//*************************************************************************************FORCE COLOR & BRIGHTNESS - LEVEL
IF sDeviceType = Domoticz_Constants.sType_LightSwitch
AND xForceSetValues
AND NOT xFading_int
	//Brightness	
AND ((NOT _Domoticz_EqualWithWindow(byBrightness_int, scColorData_Act.byBrightness, 5) AND xEnable_int)
	OR (NOT _Domoticz_EqualWithWindow(byBrightness_int, scColorData_Act.byBrightness, 1) AND (byBrightness_int = 0 OR NOT xEnable_int))) 
THEN
	
	//Set mode
	afb_ObjectArrayReal_InOut[1].eCommandType := _Domoticz_eCommandType.SetBrightness;	//Don't use default uDevice
	
	//Transfer outgoing data
	afb_ObjectArrayReal_InOut[1].arValueSet[Domoticz_eSValues_Colors.Brightness]:= _Domoticz_RoundDecimals(((TO_REAL(byBrightness_int)/255)*100),0);

	//Force
	afb_ObjectArrayReal_InOut[1].ForceSet(tForceSetValues_int);

//*************************************************************************************FORCE COLOR & BRIGHTNESS - COLOR SWITCH
ELSIF sDeviceType = Domoticz_Constants.sType_ColorSwitch
AND xForceSetValues
AND NOT xFading_int
AND (NOT xColorActValid OR NOT xEnable_int OR (xEnable_int AND NOT xEnabled))
	//Brightness	
AND ((NOT _Domoticz_EqualWithWindow(byBrightness_int, scColorData_Act.byBrightness, 5) AND xEnable_int)
	OR (NOT _Domoticz_EqualWithWindow(byBrightness_int, scColorData_Act.byBrightness, 1) AND (byBrightness_int = 0 OR NOT xEnable_int))
	//Colors
	OR (NOT _Domoticz_EqualWithWindow(scColorData_Set.byRed, scColorData_Act.byRed, 1) AND xEnable_int)
	OR (NOT _Domoticz_EqualWithWindow(scColorData_Set.byGreen, scColorData_Act.byGreen, 1) AND xEnable_int)
	OR (NOT _Domoticz_EqualWithWindow(scColorData_Set.byBlue, scColorData_Act.byBlue, 1) AND xEnable_int)
	//Temperature
	OR (NOT _Domoticz_EqualWithWindow(scColorData_Set.byColdWhite, scColorData_Act.byColdWhite, 1) AND xEnable_int)
	OR (NOT _Domoticz_EqualWithWindow(scColorData_Set.byWarmWhite, scColorData_Act.byWarmWhite, 1) AND xEnable_int)) 
THEN
	
	//Set mode
	afb_ObjectArrayReal_InOut[1].eCommandType := _Domoticz_eCommandType.SetColor;	//Don't use default uDevice
	
	//Transfer outgoing data
	afb_ObjectArrayReal_InOut[1].arValueSet[Domoticz_eSValues_Colors.Brightness]:= _Domoticz_RoundDecimals(((TO_REAL(byBrightness_int)/255)*100),0);
	afb_ObjectArrayReal_InOut[1].arValueSet[Domoticz_eSValues_Colors.Red]		:= TO_REAL(scColorData_Set.byRed);
	afb_ObjectArrayReal_InOut[1].arValueSet[Domoticz_eSValues_Colors.Green]	:= TO_REAL(scColorData_Set.byGreen);
	afb_ObjectArrayReal_InOut[1].arValueSet[Domoticz_eSValues_Colors.Blue]		:= TO_REAL(scColorData_Set.byBlue);
	afb_ObjectArrayReal_InOut[1].arValueSet[Domoticz_eSValues_Colors.ColdWhite] := TO_REAL(scColorData_Set.byColdWhite);
	afb_ObjectArrayReal_InOut[1].arValueSet[Domoticz_eSValues_Colors.WarmWhite] := TO_REAL(scColorData_Set.byWarmWhite);

	//Force
	afb_ObjectArrayReal_InOut[1].ForceSet(tForceSetValues_int);
END_IF

//*************************************************************************************ERRORS
fbEI_DataTimeOut.sInstanceName := sInstanceName;
fbEI_DataTimeOut.tErrorDelay := T#500MS;	//Give objects TIME TO be overruled BY other updates
fbEI_DataTimeOut(
	scConnector:= scConnector,
	xError:= xDataTimeOut_int
			AND (afb_ObjectArrayReal_InOut[1].xDataTimedOut),
	eErrorID:= Domoticz_eErrors.ObjectDataTimeOut
);
END_ACTION

{attribute 'monitoring' := 'call'} PROPERTY tFadeTime :TIME
GET
tFadeTime := tFadeTime_int;
END_GET
SET
tFadeTime_int := tFadeTime;
END_SET
END_PROPERTY

{attribute 'monitoring' := 'call'} PROPERTY tFadeUpdateTime :TIME
SET
tFadeUpdateTime_int := tFadeUpdateTime;
END_SET
GET
tFadeUpdateTime := tFadeUpdateTime_int;
END_GET
END_PROPERTY

{attribute 'monitoring' := 'call'} PROPERTY xFading :BOOL
GET
xFading := xFading_int;
END_GET
END_PROPERTY

END_FUNCTION_BLOCK

// Functions/_Domoticz_EqualWithWindow
{attribute 'conditionalshow_all_locals'}
{attribute 'conditionalshow'}
FUNCTION _Domoticz_EqualWithWindow :BOOL
VAR_INPUT
	rInput1, rInput2, rWindow :REAL;
END_VAR
VAR
END_VAR

_Domoticz_EqualWithWindow := (rInput1 >= (rInput2 - rWindow) AND rInput1 <= (rInput2 + rWindow));

END_FUNCTION

// Functions/_Domoticz_ColorFactor
{attribute 'conditionalshow_all_locals'}
{attribute 'conditionalshow'}
FUNCTION _Domoticz_ColorFactor :REAL
VAR_INPUT
	byColorSet	:BYTE;
	byColorAct	:BYTE;
END_VAR
VAR
END_VAR

IF byColorAct <> 0 AND byColorSet <> 0 THEN
	_Domoticz_ColorFactor := TO_REAL(byColorAct)/TO_REAL(byColorSet);
ELSIF byColorAct <> 0 AND byColorSet = 0 THEN
	_Domoticz_ColorFactor := -255;
ELSIF byColorAct = 0 AND byColorSet <> 0 THEN
	_Domoticz_ColorFactor := 255;
ELSE
	_Domoticz_ColorFactor := 0;
END_IF

END_FUNCTION

// Function Blocks/Hardware/Weather/Domoticz_AccuWeather
{attribute 'conditionalshow_all_locals'}
FUNCTION_BLOCK Domoticz_AccuWeather EXTENDS _Domoticz_Connector_Out
VAR_INPUT
	uiIdentifier_TempHumBaro	:UINT;	//Temperature/humidity/barometer
	uiIdentifier_Rain			:UINT;	//Rain rate and actual
	uiIdentifier_Wind			:UINT;	//Wind (direction,strenght)
	uiIdentifier_Visibility		:UINT;	//Visibility outside
	uiIdentifier_UV				:UINT;	//UV power
END_VAR
VAR_OUTPUT
	rTemperature				:REAL;
	rDewPoint					:REAL;
	rChill						:REAL;
	rHumidity					:REAL;
	rBaroMeter					:REAL;
	rRain						:REAL;
	rRainRate					:REAL;
	rWindSpeed					:REAL;
	rWindGust					:REAL;
	rWindDirection				:REAL;
	rVisibility					:REAL;
	rUV							:REAL;
END_VAR
VAR
	afb_ObjectArrayReal_Out		:ARRAY[1..3] OF _Domoticz_ObjectArrayReal_Out;
	afb_ObjectReal_Out			:ARRAY[1..2] OF _Domoticz_ObjectReal_Out;
END_VAR

IF __ISVALIDREF(scConnector) THEN
	Main();
END_IF

ACTION Main:
{attribute 'conditionalshow'}
//Call parent function
SUPER^.Main();

//Call all functions
//Extended data timeout (Weather not updated frequently)
afb_ObjectArrayReal_Out[1].tDataTimeOut := T#24H;
afb_ObjectArrayReal_Out[1](	scConnector := scConnector, 	uiIdentifier := uiIdentifier_TempHumBaro,	rxUpdateInterlock := rxUpdateInterlock_int);
                                                            
afb_ObjectArrayReal_Out[2].tDataTimeOut := T#24H;           
afb_ObjectArrayReal_Out[2](	scConnector := scConnector, 	uiIdentifier := uiIdentifier_Wind,			rxUpdateInterlock := rxUpdateInterlock_int);
                                                            
afb_ObjectArrayReal_Out[3].tDataTimeOut := T#24H;           
afb_ObjectArrayReal_Out[3](	scConnector := scConnector,		uiIdentifier := uiIdentifier_Rain,			rxUpdateInterlock := rxUpdateInterlock_int);
                                                            
afb_ObjectReal_Out[1].tDataTimeOut := T#24H;                
afb_ObjectReal_Out[1](		scConnector := scConnector, 	uiIdentifier := uiIdentifier_Visibility,	rxUpdateInterlock := rxUpdateInterlock_int,		rValueAct => rVisibility);
                                                            
afb_ObjectReal_Out[2].tDataTimeOut := T#24H;                
afb_ObjectReal_Out[2](		scConnector := scConnector, 	uiIdentifier := uiIdentifier_UV,			rxUpdateInterlock := rxUpdateInterlock_int,		rValueAct => rUV);

//Output arrays
rTemperature 	:= afb_ObjectArrayReal_Out[1].arValueAct[Domoticz_eSValues_TempHumBaro.Temperature];
rDewPoint		:= afb_ObjectArrayReal_Out[1].arValueAct[Domoticz_eSValues_TempHumBaro.DewPoint];
rHumidity		:= afb_ObjectArrayReal_Out[1].arValueAct[Domoticz_eSValues_TempHumBaro.Humidity];
rBaroMeter		:= afb_ObjectArrayReal_Out[1].arValueAct[Domoticz_eSValues_TempHumBaro.Barometer];

rWindSpeed	 	:= afb_ObjectArrayReal_Out[2].arValueAct[Domoticz_eSValues_Wind.Speed];
rChill			:= afb_ObjectArrayReal_Out[2].arValueAct[Domoticz_eSValues_Wind.Chill];
rWindGust		:= afb_ObjectArrayReal_Out[2].arValueAct[Domoticz_eSValues_Wind.Gust];
rWindDirection	:= afb_ObjectArrayReal_Out[2].arValueAct[Domoticz_eSValues_Wind.Bearing];

rRain		 	:= afb_ObjectArrayReal_Out[3].arValueAct[Domoticz_eSValues_Rain.Rain];
rRainRate		:= afb_ObjectArrayReal_Out[3].arValueAct[Domoticz_eSValues_Rain.RainRate];

//Errors
fbEI_DataTimeOut.sInstanceName := sInstanceName;
fbEI_DataTimeOut.tErrorDelay := T#500MS;	//Give objects TIME TO be overruled BY other updates
fbEI_DataTimeOut(
	scConnector:= scConnector,
	xError:= xDataTimeOut_int
			AND (afb_ObjectArrayReal_Out[1].xDataTimedOut
			OR afb_ObjectArrayReal_Out[2].xDataTimedOut
			OR afb_ObjectArrayReal_Out[3].xDataTimedOut
			OR afb_ObjectReal_Out[1].xDataTimedOut
			OR afb_ObjectReal_Out[2].xDataTimedOut),
	eErrorID:= Domoticz_eErrors.ObjectDataTimeOut
);
END_ACTION

END_FUNCTION_BLOCK

// Function Blocks/Hardware/Weather/Domoticz_BuienAlarm
{attribute 'conditionalshow_all_locals'}
FUNCTION_BLOCK Domoticz_BuienAlarm EXTENDS _Domoticz_Connector_Out
VAR_INPUT
	uiIdentifier_Rain			:UINT;	//Rain rate and actual
	uiIdentifier_RainAlert		:UINT;	//Rain alert
	uiIdentifier_RainForecast	:UINT;	//Rain forecast
END_VAR
VAR_OUTPUT
	rRain						:REAL;
	rRainRate					:REAL;
	rRainForecast				:REAL;
	sRainAlert					:STRING(Domoticz_Constants.uiMaxSValuesize);
	sRainForecast				:STRING(Domoticz_Constants.uiMaxSValuesize);
END_VAR
VAR
	afb_ObjectArrayReal_Out		:ARRAY[1..1] OF _Domoticz_ObjectArrayReal_Out;
	afb_ObjectString_Out		:ARRAY[1..2] OF _Domoticz_ObjectString_Out;
END_VAR

IF __ISVALIDREF(scConnector) THEN
	Main();
END_IF

ACTION Main:
{attribute 'conditionalshow'}
//Call parent function
SUPER^.Main();

//Call all functions
//Extended data timeout, expect a litle rain at least once every two weeks.
afb_ObjectArrayReal_Out[1].tDataTimeOut := T#14D;
afb_ObjectArrayReal_Out[1].eDataSource := _Domoticz_eDataSource.HTTP;  
afb_ObjectArrayReal_Out[1](	scConnector := scConnector, 	uiIdentifier := uiIdentifier_Rain,			rxUpdateInterlock := rxUpdateInterlock_int);
                                                                                                                                                                                  
afb_ObjectString_Out[1].tDataTimeOut := T#14D;      
afb_ObjectString_Out[1].eDataSource := _Domoticz_eDataSource.HTTP;                                                                              
afb_ObjectString_Out[1](	scConnector := scConnector, 	uiIdentifier := uiIdentifier_RainAlert, 	rxUpdateInterlock := rxUpdateInterlock_int,			sValueAct => sRainAlert);
                                                                                                                                                                                
afb_ObjectString_Out[2].tDataTimeOut := T#14D; 
afb_ObjectString_Out[2].eDataSource := _Domoticz_eDataSource.HTTP;                                                                                                              
afb_ObjectString_Out[2](	scConnector := scConnector, 	uiIdentifier := uiIdentifier_RainForecast, 	rxUpdateInterlock := rxUpdateInterlock_int,			sValueAct => sRainForecast);

//Output arrays
rRain		 	:= afb_ObjectArrayReal_Out[1].arValueAct[Domoticz_eSValues_Rain.Rain];
rRainRate		:= afb_ObjectArrayReal_Out[1].arValueAct[Domoticz_eSValues_Rain.RainRate];
rRainForecast	:= _Domoticz_StringToReal(sRainAlert);

//Errors
fbEI_DataTimeOut.sInstanceName := sInstanceName;
fbEI_DataTimeOut.tErrorDelay := T#500MS;	//Give objects TIME TO be overruled BY other updates
fbEI_DataTimeOut(
	scConnector:= scConnector,
	xError:= xDataTimeOut_int
			AND (afb_ObjectArrayReal_Out[1].xDataTimedOut
			OR afb_ObjectString_Out[1].xDataTimedOut
			OR afb_ObjectString_Out[2].xDataTimedOut),
	eErrorID:= Domoticz_eErrors.ObjectDataTimeOut
);
END_ACTION

END_FUNCTION_BLOCK

// Function Blocks/Hardware/Weather/Domoticz_BuienRadar
{attribute 'conditionalshow_all_locals'}
FUNCTION_BLOCK Domoticz_BuienRadar EXTENDS _Domoticz_Connector_Out
VAR_INPUT
	uiIdentifier_TempHumBaro		:UINT;	//Temperature/humidity/barometer
	uiIdentifier_TempGround			:UINT;	//Ground temperature
	uiIdentifier_TempFeel			:UINT;	//Feel temperature
	uiIdentifier_Wind				:UINT;	//Wind (direction,strenght)	
	uiIdentifier_Visibility			:UINT;	//Visibility outside
	uiIdentifier_Solar				:UINT;	//Solar power
	uiIdentifier_Rain				:UINT;	//Rain
	uiIdentifier_RainNextHour		:UINT;	//Rain forecast next hour
	uiIdentifier_RainIntensity		:UINT;	//Rain intensity
	uiIdentifier_RainingMeasured	:UINT;	//Raining - measured at weather station
	uiIdentifier_RainingForecast	:UINT;	//Raining - forecasted at current location
	uiIdentifier_NextRainTime		:UINT;	//Next rainshower time
	uiIdentifier_NextRainDuration	:UINT;	//Next rainshower duration
	uiIdentifier_NextRainAvgRate	:UINT;	//Next rainshower avg rate
	uiIdentifier_NextRainMaxRate	:UINT;	//Next rainshower max rate
END_VAR
VAR_OUTPUT
	rTemperature					:REAL;
	rTemperatureGround				:REAL;
	rTemperatureFeel				:REAL;
	rHumidity						:REAL;
	rBaroMeter						:REAL;
	rWindSpeed						:REAL;
	rWindGust						:REAL;
	rWindDirection					:REAL;
	rVisibility						:REAL;
	rSolar							:REAL;
	rRain							:REAL;
	rRainRate						:REAL;
	rRainNextHour					:REAL;
	rRainIntensity					:REAL;
	xRainingMeasured				:BOOL;
	xRainingForecast				:BOOL;
	tNextRainTime					:TIME;
	tNextRainDuration				:TIME;
	rNextRainAvgRate				:REAL;
	rNextRainMaxRate				:REAL;
END_VAR                         	
VAR                             	
	afb_ObjectArrayReal_Out			:ARRAY[1..3] OF _Domoticz_ObjectArrayReal_Out;
	afb_ObjectReal_Out				:ARRAY[1..10] OF _Domoticz_ObjectReal_Out;
	afb_ObjectBool_Out				:ARRAY[1..2] OF _Domoticz_ObjectBool_Out;
END_VAR

IF __ISVALIDREF(scConnector) THEN
	Main();
END_IF

ACTION Main:
{attribute 'conditionalshow'}
//Call parent function
SUPER^.Main();

//Call all functions
//Extended data timeout (Weather not updated frequently)
afb_ObjectArrayReal_Out[1].tDataTimeOut := T#24H;
afb_ObjectArrayReal_Out[1].eDataSource := _Domoticz_eDataSource.HTTP;
afb_ObjectArrayReal_Out[1](	scConnector := scConnector, 	uiIdentifier := uiIdentifier_TempHumBaro,		rxUpdateInterlock := rxUpdateInterlock_int);
                                                                                                                                                
afb_ObjectArrayReal_Out[2].tDataTimeOut := T#24H;    
afb_ObjectArrayReal_Out[2].eDataSource := _Domoticz_eDataSource.HTTP;                                                                                           
afb_ObjectArrayReal_Out[2](	scConnector := scConnector, 	uiIdentifier := uiIdentifier_Rain,				rxUpdateInterlock := rxUpdateInterlock_int);
                                                                                             
afb_ObjectArrayReal_Out[3].tDataTimeOut := T#24H;                                            
afb_ObjectArrayReal_Out[3].eDataSource := _Domoticz_eDataSource.HTTP;                                 
afb_ObjectArrayReal_Out[3](	scConnector := scConnector, 	uiIdentifier := uiIdentifier_Wind,				rxUpdateInterlock := rxUpdateInterlock_int);
                                                                                                                                                
afb_ObjectReal_Out[1].tDataTimeOut := T#24H;  
afb_ObjectReal_Out[1].eDataSource := _Domoticz_eDataSource.HTTP;                                                                                                  
afb_ObjectReal_Out[1](		scConnector := scConnector, 	uiIdentifier := uiIdentifier_TempGround,		rxUpdateInterlock := rxUpdateInterlock_int,			rValueAct => rTemperatureGround);
                                                                                                                                            
afb_ObjectReal_Out[2].tDataTimeOut := T#24H;                                                                                                
afb_ObjectReal_Out[2].eDataSource := _Domoticz_eDataSource.HTTP;                                                                                           
afb_ObjectReal_Out[2](		scConnector := scConnector, 	uiIdentifier := uiIdentifier_TempFeel,			rxUpdateInterlock := rxUpdateInterlock_int,			rValueAct => rTemperatureFeel);
                                                                                                                                            
afb_ObjectReal_Out[3].tDataTimeOut := T#24H;                                                                                                
afb_ObjectReal_Out[3].eDataSource := _Domoticz_eDataSource.HTTP;                                                                                           
afb_ObjectReal_Out[3](		scConnector := scConnector, 	uiIdentifier := uiIdentifier_Visibility,		rxUpdateInterlock := rxUpdateInterlock_int,			rValueAct => rVisibility);
                                                                                                                                            
afb_ObjectReal_Out[4].tDataTimeOut := T#24H;                                                                                                
afb_ObjectReal_Out[4].eDataSource := _Domoticz_eDataSource.HTTP;                                                                                               
afb_ObjectReal_Out[4](		scConnector := scConnector, 	uiIdentifier := uiIdentifier_Solar,				rxUpdateInterlock := rxUpdateInterlock_int,			rValueAct => rSolar);
                                                                                                                                            
afb_ObjectReal_Out[5].tDataTimeOut := T#24H;                                                                                                
afb_ObjectReal_Out[5].eDataSource := _Domoticz_eDataSource.HTTP;                                                                                              
afb_ObjectReal_Out[5](		scConnector := scConnector, 	uiIdentifier := uiIdentifier_RainNextHour,		rxUpdateInterlock := rxUpdateInterlock_int,			rValueAct => rRainNextHour);
                                                                                                                                            
afb_ObjectReal_Out[6].tDataTimeOut := T#24H;                                                                                                
afb_ObjectReal_Out[6].eDataSource := _Domoticz_eDataSource.HTTP;                                                                                              
afb_ObjectReal_Out[6](		scConnector := scConnector, 	uiIdentifier := uiIdentifier_RainIntensity,		rxUpdateInterlock := rxUpdateInterlock_int,			rValueAct => rRainIntensity);
                                                                                                                                                                                           
afb_ObjectReal_Out[7].tDataTimeOut := T#24H;      
afb_ObjectReal_Out[7].eDataSource := _Domoticz_eDataSource.HTTP;                                                                                                                                         
afb_ObjectReal_Out[7](		scConnector := scConnector, 	uiIdentifier := uiIdentifier_NextRainTime,		rxUpdateInterlock := rxUpdateInterlock_int);                             
                                                                                                                                           
afb_ObjectReal_Out[8].tDataTimeOut := T#24H;                                                                
afb_ObjectReal_Out[8].eDataSource := _Domoticz_eDataSource.HTTP;                                                                                          
afb_ObjectReal_Out[8](		scConnector := scConnector, 	uiIdentifier := uiIdentifier_NextRainDuration,	rxUpdateInterlock := rxUpdateInterlock_int);                             
                                                                                                                                                                                           
afb_ObjectReal_Out[9].tDataTimeOut := T#24H;                                                                                                                                               
afb_ObjectReal_Out[9].eDataSource := _Domoticz_eDataSource.HTTP;
afb_ObjectReal_Out[9](		scConnector := scConnector, 	uiIdentifier := uiIdentifier_NextRainAvgRate,	rxUpdateInterlock := rxUpdateInterlock_int,			rValueAct => rNextRainAvgRate);
                                                                                                                                         
afb_ObjectReal_Out[10].tDataTimeOut := T#24H;                                                                                            
afb_ObjectReal_Out[10].eDataSource := _Domoticz_eDataSource.HTTP;                                                                                        
afb_ObjectReal_Out[10](		scConnector := scConnector, 	uiIdentifier := uiIdentifier_NextRainMaxRate,	rxUpdateInterlock := rxUpdateInterlock_int,			rValueAct => rNextRainMaxRate);
                                                                                                                                         
afb_ObjectBool_Out[1].tDataTimeOut := T#24H;                                                                                             
afb_ObjectBool_Out[1].eDataSource := _Domoticz_eDataSource.HTTP;                                                                          
afb_ObjectBool_Out[1](		scConnector := scConnector, 	uiIdentifier := uiIdentifier_RainingMeasured,	rxUpdateInterlock := rxUpdateInterlock_int,			xValueAct => xRainingMeasured);
                                                                                                                                         
afb_ObjectBool_Out[2].tDataTimeOut := T#14D;                                                                                             
afb_ObjectBool_Out[2].eDataSource := _Domoticz_eDataSource.HTTP;                                                                                
afb_ObjectBool_Out[2](		scConnector := scConnector, 	uiIdentifier := uiIdentifier_RainingForecast,	rxUpdateInterlock := rxUpdateInterlock_int,			xValueAct => xRainingForecast);


//Output arrays
rTemperature 		:= afb_ObjectArrayReal_Out[1].arValueAct[Domoticz_eSValues_TempHumBaro.Temperature];
rHumidity			:= afb_ObjectArrayReal_Out[1].arValueAct[Domoticz_eSValues_TempHumBaro.Humidity];
rBaroMeter			:= afb_ObjectArrayReal_Out[1].arValueAct[Domoticz_eSValues_TempHumBaro.Barometer];
                		                	
rRain		 		:= afb_ObjectArrayReal_Out[2].arValueAct[Domoticz_eSValues_Rain.Rain];
rRainRate			:= afb_ObjectArrayReal_Out[2].arValueAct[Domoticz_eSValues_Rain.RainRate];

rWindSpeed	 		:= afb_ObjectArrayReal_Out[3].arValueAct[Domoticz_eSValues_Wind.Speed];
rWindGust			:= afb_ObjectArrayReal_Out[3].arValueAct[Domoticz_eSValues_Wind.Gust];
rWindDirection		:= afb_ObjectArrayReal_Out[3].arValueAct[Domoticz_eSValues_Wind.Bearing];
                	
tNextRainTime		:= TO_TIME(afb_ObjectReal_Out[7].rValueAct * 60 * 1000);
tNextRainDuration 	:= TO_TIME(afb_ObjectReal_Out[8].rValueAct * 60 * 1000); 
										   
//Errors
fbEI_DataTimeOut.sInstanceName := sInstanceName;
fbEI_DataTimeOut.tErrorDelay := T#500MS;	//Give objects TIME TO be overruled BY other updates
fbEI_DataTimeOut(
	scConnector:= scConnector,
	xError:= xDataTimeOut_int
			AND (afb_ObjectArrayReal_Out[1].xDataTimedOut
			OR afb_ObjectArrayReal_Out[2].xDataTimedOut
			OR afb_ObjectArrayReal_Out[3].xDataTimedOut
			OR afb_ObjectReal_Out[1].xDataTimedOut
			OR afb_ObjectReal_Out[2].xDataTimedOut
			OR afb_ObjectReal_Out[3].xDataTimedOut
			OR afb_ObjectReal_Out[4].xDataTimedOut
			OR afb_ObjectReal_Out[5].xDataTimedOut
			OR afb_ObjectReal_Out[6].xDataTimedOut
			OR afb_ObjectReal_Out[7].xDataTimedOut
			OR afb_ObjectReal_Out[8].xDataTimedOut
			OR afb_ObjectReal_Out[9].xDataTimedOut
			OR afb_ObjectReal_Out[10].xDataTimedOut
			OR afb_ObjectBool_Out[1].xDataTimedOut
			OR afb_ObjectBool_Out[2].xDataTimedOut),
	eErrorID:= Domoticz_eErrors.ObjectDataTimeOut
);
END_ACTION

END_FUNCTION_BLOCK

// Function Blocks/Hardware/Weather/Domoticz_BuienRadar_Forecast
{attribute 'conditionalshow_all_locals'}
FUNCTION_BLOCK Domoticz_BuienRadar_Forecast EXTENDS _Domoticz_Connector_Out
VAR_INPUT
	uiIdentifier_TempMin		:UINT;	//Minimal temperature
	uiIdentifier_TempMax		:UINT;	//Maixmal temperature
	uiIdentifier_SunChance		:UINT;	//Chance for sunshine (%)
	uiIdentifier_RainChance		:UINT;	//Chance for rain (%)
	uiIdentifier_RainAmount		:UINT;	//Rain amount for whole day
	uiIdentifier_SnowAmount		:UINT;	//Snow amount for whole day
END_VAR
VAR_OUTPUT
	rTemperatureMin				:REAL;
	rTemperatureMax				:REAL;
	iSunChance					:INT;
	iRainChance					:INT;
	rRainAmount					:REAL;
	rSnowAmount					:REAL;
END_VAR
VAR
	afb_ObjectReal_Out			:ARRAY[1..6] OF _Domoticz_ObjectReal_Out;
END_VAR

IF __ISVALIDREF(scConnector) THEN
	Main();
END_IF

ACTION Main:
{attribute 'conditionalshow'}
//Call parent function
SUPER^.Main();

//Call all functions
//Extended data timeout (Weather not updated frequently)
afb_ObjectReal_Out[1].tDataTimeOut := T#36H;
afb_ObjectReal_Out[1].eDataSource := _Domoticz_eDataSource.HTTP;
afb_ObjectReal_Out[1](	scConnector := scConnector, 	uiIdentifier := uiIdentifier_TempMin,		rxUpdateInterlock := rxUpdateInterlock_int,			rValueAct => rTemperatureMin);
                                                            
afb_ObjectReal_Out[2].tDataTimeOut := T#36H;
afb_ObjectReal_Out[2].eDataSource := _Domoticz_eDataSource.HTTP;            
afb_ObjectReal_Out[2](	scConnector := scConnector, 	uiIdentifier := uiIdentifier_TempMax,		rxUpdateInterlock := rxUpdateInterlock_int,			rValueAct => rTemperatureMax);
                                                            
afb_ObjectReal_Out[3].tDataTimeOut := T#36H;
afb_ObjectReal_Out[3].eDataSource := _Domoticz_eDataSource.HTTP;          
afb_ObjectReal_Out[3](	scConnector := scConnector, 	uiIdentifier := uiIdentifier_SunChance,		rxUpdateInterlock := rxUpdateInterlock_int);
                                                            
afb_ObjectReal_Out[4].tDataTimeOut := T#36H;
afb_ObjectReal_Out[4].eDataSource := _Domoticz_eDataSource.HTTP;            
afb_ObjectReal_Out[4](	scConnector := scConnector, 	uiIdentifier := uiIdentifier_RainChance,	rxUpdateInterlock := rxUpdateInterlock_int);
                                                            
afb_ObjectReal_Out[4].tDataTimeOut := T#36H;
afb_ObjectReal_Out[4].eDataSource := _Domoticz_eDataSource.HTTP;              
afb_ObjectReal_Out[5](	scConnector := scConnector, 	uiIdentifier := uiIdentifier_RainAmount,	rxUpdateInterlock := rxUpdateInterlock_int,			rValueAct => rRainAmount);
                                                            
afb_ObjectReal_Out[6].tDataTimeOut := T#36H;
afb_ObjectReal_Out[6].eDataSource := _Domoticz_eDataSource.HTTP;             
afb_ObjectReal_Out[6](	scConnector := scConnector, 	uiIdentifier := uiIdentifier_SnowAmount,	rxUpdateInterlock := rxUpdateInterlock_int,			rValueAct => rSnowAmount);

//Output other data types
iSunChance := TO_INT(afb_ObjectReal_Out[3].rValueAct);
iRainChance := TO_INT(afb_ObjectReal_Out[4].rValueAct);

//Errors
fbEI_DataTimeOut.sInstanceName := sInstanceName;
fbEI_DataTimeOut.tErrorDelay := T#500MS;	//Give objects TIME TO be overruled BY other updates
fbEI_DataTimeOut(
	scConnector:= scConnector,
	xError:= xDataTimeOut_int
			AND (afb_ObjectReal_Out[1].xDataTimedOut
			OR afb_ObjectReal_Out[2].xDataTimedOut
			OR afb_ObjectReal_Out[3].xDataTimedOut
			OR afb_ObjectReal_Out[4].xDataTimedOut
			OR afb_ObjectReal_Out[5].xDataTimedOut
			OR afb_ObjectReal_Out[6].xDataTimedOut),
	eErrorID:= Domoticz_eErrors.ObjectDataTimeOut
);
END_ACTION

END_FUNCTION_BLOCK

// Function Blocks/Hardware/Weather/Domoticz_DarkSky
{attribute 'conditionalshow_all_locals'}
FUNCTION_BLOCK Domoticz_DarkSky EXTENDS _Domoticz_Connector_Out
VAR_INPUT
	uiIdentifier_TempHumBaro	:UINT;	//Temperature/humidity/barometer
	uiIdentifier_Rain			:UINT;	//Rain rate and actual
	uiIdentifier_Wind			:UINT;	//Wind (direction,strenght)
	uiIdentifier_Visibility		:UINT;	//Visibility outside
	uiIdentifier_UV				:UINT;	//UV power
	uiIdentifier_Ozone			:UINT;	//Ozone level
END_VAR
VAR_OUTPUT
	rTemperature				:REAL;
	rDewPoint					:REAL;
	rChill						:REAL;
	rHumidity					:REAL;
	rBaroMeter					:REAL;
	rRain						:REAL;
	rRainRate					:REAL;
	rWindSpeed					:REAL;
	rWindGust					:REAL;
	rWindDirection				:REAL;
	rVisibility					:REAL;
	rUV							:REAL;
	rOzone						:REAL;
END_VAR
VAR
	afb_ObjectArrayReal_Out		:ARRAY[1..3] OF _Domoticz_ObjectArrayReal_Out;
	afb_ObjectReal_Out			:ARRAY[1..3] OF _Domoticz_ObjectReal_Out;
END_VAR

IF __ISVALIDREF(scConnector) THEN
	Main();
END_IF

ACTION Main:
{attribute 'conditionalshow'}
//Call parent function
SUPER^.Main();

//Call all functions
//Extended data timeout (Weather not updated frequently)
afb_ObjectArrayReal_Out[1].tDataTimeOut := T#24H;
afb_ObjectArrayReal_Out[1].eDataSource := _Domoticz_eDataSource.HTTP;
afb_ObjectArrayReal_Out[1](	scConnector := scConnector, 	uiIdentifier := uiIdentifier_TempHumBaro,	rxUpdateInterlock := rxUpdateInterlock_int);

afb_ObjectArrayReal_Out[2].tDataTimeOut := T#24H;
afb_ObjectArrayReal_Out[2].eDataSource := _Domoticz_eDataSource.HTTP;
afb_ObjectArrayReal_Out[2](	scConnector := scConnector, 	uiIdentifier := uiIdentifier_Wind,			rxUpdateInterlock := rxUpdateInterlock_int);

afb_ObjectArrayReal_Out[2].tDataTimeOut := T#24H;
afb_ObjectArrayReal_Out[2].eDataSource := _Domoticz_eDataSource.HTTP;
afb_ObjectArrayReal_Out[3](	scConnector := scConnector, 	uiIdentifier := uiIdentifier_Rain,			rxUpdateInterlock := rxUpdateInterlock_int);

afb_ObjectReal_Out[1].tDataTimeOut := T#24H;
afb_ObjectReal_Out[1].eDataSource := _Domoticz_eDataSource.HTTP;
afb_ObjectReal_Out[1](		scConnector := scConnector, 	uiIdentifier := uiIdentifier_Visibility,	rxUpdateInterlock := rxUpdateInterlock_int,			rValueAct => rVisibility);
                                                            
afb_ObjectReal_Out[2].tDataTimeOut := T#24H;                
afb_ObjectReal_Out[2].eDataSource := _Domoticz_eDataSource.HTTP;
afb_ObjectReal_Out[2](		scConnector := scConnector, 	uiIdentifier := uiIdentifier_UV,			rxUpdateInterlock := rxUpdateInterlock_int,			rValueAct => rUV);
                                                            
afb_ObjectReal_Out[3].tDataTimeOut := T#24H;                
afb_ObjectReal_Out[3].eDataSource := _Domoticz_eDataSource.HTTP;
afb_ObjectReal_Out[3](		scConnector := scConnector, 	uiIdentifier := uiIdentifier_Ozone,			rxUpdateInterlock := rxUpdateInterlock_int,			rValueAct => rOzone);

//Output arrays
rTemperature 	:= afb_ObjectArrayReal_Out[1].arValueAct[Domoticz_eSValues_TempHumBaro.Temperature];
rDewPoint		:= afb_ObjectArrayReal_Out[1].arValueAct[Domoticz_eSValues_TempHumBaro.DewPoint];
rHumidity		:= afb_ObjectArrayReal_Out[1].arValueAct[Domoticz_eSValues_TempHumBaro.Humidity];
rBaroMeter		:= afb_ObjectArrayReal_Out[1].arValueAct[Domoticz_eSValues_TempHumBaro.Barometer];

rWindSpeed	 	:= afb_ObjectArrayReal_Out[2].arValueAct[Domoticz_eSValues_Wind.Speed];
rChill			:= afb_ObjectArrayReal_Out[2].arValueAct[Domoticz_eSValues_Wind.Chill];
rWindGust		:= afb_ObjectArrayReal_Out[2].arValueAct[Domoticz_eSValues_Wind.Gust];
rWindDirection	:= afb_ObjectArrayReal_Out[2].arValueAct[Domoticz_eSValues_Wind.Bearing];

rRain		 	:= afb_ObjectArrayReal_Out[3].arValueAct[Domoticz_eSValues_Rain.Rain];
rRainRate		:= afb_ObjectArrayReal_Out[3].arValueAct[Domoticz_eSValues_Rain.RainRate];
											
//Errors
fbEI_DataTimeOut.sInstanceName := sInstanceName;
fbEI_DataTimeOut.tErrorDelay := T#500MS;	//Give objects TIME TO be overruled BY other updates
fbEI_DataTimeOut(
	scConnector:= scConnector,
	xError:= xDataTimeOut_int
			AND (afb_ObjectArrayReal_Out[1].xDataTimedOut
			OR afb_ObjectArrayReal_Out[2].xDataTimedOut
			OR afb_ObjectArrayReal_Out[3].xDataTimedOut
			OR afb_ObjectReal_Out[1].xDataTimedOut
			OR afb_ObjectReal_Out[2].xDataTimedOut
			OR afb_ObjectReal_Out[3].xDataTimedOut),
	eErrorID:= Domoticz_eErrors.ObjectDataTimeOut
);
END_ACTION

END_FUNCTION_BLOCK

// Function Blocks/Hardware/Weather/Domoticz_OpenWeatherMap
{attribute 'conditionalshow_all_locals'}
FUNCTION_BLOCK Domoticz_OpenWeatherMap EXTENDS _Domoticz_Connector_Out
VAR_INPUT
	uiIdentifier_TempHumBaro	:UINT;	//Temperature/humidity/barometer
	uiIdentifier_Rain			:UINT;	//Rain rate and actual
	uiIdentifier_Wind			:UINT;	//Wind (direction,strenght)
	uiIdentifier_Visibility		:UINT;	//Visibility outside
	uiIdentifier_Cloudiness		:UINT;	//UV power
END_VAR
VAR_OUTPUT
	rTemperature				:REAL;
	rDewPoint					:REAL;
	rChill						:REAL;
	rHumidity					:REAL;
	rBaroMeter					:REAL;
	rRain						:REAL;
	rWindSpeed					:REAL;
	rWindGust					:REAL;
	rWindDirection				:REAL;
	rVisibility					:REAL;
	rCloudiness					:REAL;
END_VAR
VAR
	afb_ObjectArrayReal_Out		:ARRAY[1..2] OF _Domoticz_ObjectArrayReal_Out;
	afb_ObjectReal_Out			:ARRAY[1..3] OF _Domoticz_ObjectReal_Out;
END_VAR

IF __ISVALIDREF(scConnector) THEN
	Main();
END_IF

ACTION Main:
{attribute 'conditionalshow'}
//Call parent function
SUPER^.Main();

//Call all functions
//Extended data timeout (Weather not updated frequently)
afb_ObjectArrayReal_Out[1].tDataTimeOut := T#24H;
afb_ObjectArrayReal_Out[1].eDataSource := _Domoticz_eDataSource.HTTP;
afb_ObjectArrayReal_Out[1](	scConnector := scConnector, 	uiIdentifier := uiIdentifier_TempHumBaro,	rxUpdateInterlock := rxUpdateInterlock_int);

afb_ObjectArrayReal_Out[2].tDataTimeOut := T#24H;
afb_ObjectArrayReal_Out[2].eDataSource := _Domoticz_eDataSource.HTTP;
afb_ObjectArrayReal_Out[2](	scConnector := scConnector, 	uiIdentifier := uiIdentifier_Wind,			rxUpdateInterlock := rxUpdateInterlock_int);
                                                            
afb_ObjectReal_Out[1].tDataTimeOut := T#24H;
afb_ObjectReal_Out[1].eDataSource := _Domoticz_eDataSource.HTTP;
afb_ObjectReal_Out[1](		scConnector := scConnector, 	uiIdentifier := uiIdentifier_Rain,			rxUpdateInterlock := rxUpdateInterlock_int,			rValueAct => rRain);

afb_ObjectReal_Out[2].tDataTimeOut := T#24H;
afb_ObjectReal_Out[2].eDataSource := _Domoticz_eDataSource.HTTP;
afb_ObjectReal_Out[2](		scConnector := scConnector, 	uiIdentifier := uiIdentifier_Visibility,	rxUpdateInterlock := rxUpdateInterlock_int,			rValueAct => rVisibility);

afb_ObjectReal_Out[3].tDataTimeOut := T#24H;
afb_ObjectReal_Out[3].eDataSource := _Domoticz_eDataSource.HTTP;
afb_ObjectReal_Out[3](		scConnector := scConnector, 	uiIdentifier := uiIdentifier_Cloudiness,	rxUpdateInterlock := rxUpdateInterlock_int,			rValueAct => rCloudiness);

//Output arrays
rTemperature 	:= afb_ObjectArrayReal_Out[1].arValueAct[Domoticz_eSValues_TempHumBaro.Temperature];
rDewPoint		:= afb_ObjectArrayReal_Out[1].arValueAct[Domoticz_eSValues_TempHumBaro.DewPoint];
rHumidity		:= afb_ObjectArrayReal_Out[1].arValueAct[Domoticz_eSValues_TempHumBaro.Humidity];
rBaroMeter		:= afb_ObjectArrayReal_Out[1].arValueAct[Domoticz_eSValues_TempHumBaro.Barometer];

rWindSpeed	 	:= afb_ObjectArrayReal_Out[2].arValueAct[Domoticz_eSValues_Wind.Speed];
rChill			:= afb_ObjectArrayReal_Out[2].arValueAct[Domoticz_eSValues_Wind.Chill];
rWindGust		:= afb_ObjectArrayReal_Out[2].arValueAct[Domoticz_eSValues_Wind.Gust];
rWindDirection	:= afb_ObjectArrayReal_Out[2].arValueAct[Domoticz_eSValues_Wind.Bearing];
											
//Errors
fbEI_DataTimeOut.sInstanceName := sInstanceName;
fbEI_DataTimeOut.tErrorDelay := T#500MS;	//Give objects TIME TO be overruled BY other updates
fbEI_DataTimeOut(
	scConnector:= scConnector,
	xError:= xDataTimeOut_int
			AND (afb_ObjectArrayReal_Out[1].xDataTimedOut
			OR afb_ObjectArrayReal_Out[2].xDataTimedOut
			OR afb_ObjectReal_Out[1].xDataTimedOut
			OR afb_ObjectReal_Out[2].xDataTimedOut
			OR afb_ObjectReal_Out[3].xDataTimedOut),
	eErrorID:= Domoticz_eErrors.ObjectDataTimeOut
);
END_ACTION

END_FUNCTION_BLOCK

// Function Blocks/Hardware/Weather/Domoticz_SunMoon
{attribute 'conditionalshow_all_locals'}
FUNCTION_BLOCK Domoticz_SunMoon EXTENDS _Domoticz_Connector_Out
VAR_INPUT
	uiIdentifier_SunAzimuth		:UINT;	//Sun
	uiIdentifier_SunAltitude	:UINT;	//Sun height
	uiIdentifier_SunDistance	:UINT;	//Sun distance to earth
	uiIdentifier_MoonAzimuth	:UINT;	//Moon
	uiIdentifier_MoonAltitude	:UINT;	//Moon height
	uiIdentifier_MoonDistance	:UINT;	//Moon distance to earth
	uiIdentifier_MoonPhase		:UINT;	//Moon visibility
END_VAR
VAR_OUTPUT
	rSunAzimuth					:REAL;	//Sun
	rSunAltitude				:REAL;	//Sun height
	rSunDistance				:REAL;	//Sun distance to earth
	rMoonAzimuth				:REAL;	//Moon
	rMoonAltitude				:REAL;	//Moon height
	rMoonDistance				:REAL;	//Moon distance to earth
	rMoonPhase					:REAL;	//Moon visibility
END_VAR
VAR
	afb_ObjectReal_Out				:ARRAY[1..7] OF _Domoticz_ObjectReal_Out;
END_VAR

IF __ISVALIDREF(scConnector) THEN
	Main();
END_IF

ACTION Main:
{attribute 'conditionalshow'}
//Call parent function
SUPER^.Main();

//Call all functions
//Extended data timeout (Weather not updated frequently)
afb_ObjectReal_Out[1].tDataTimeOut := T#24H;
afb_ObjectReal_Out[1].eDataSource := _Domoticz_eDataSource.HTTP;
afb_ObjectReal_Out[1](scConnector := scConnector, 	uiIdentifier := uiIdentifier_SunAzimuth,	rxUpdateInterlock := rxUpdateInterlock_int,			rValueAct => rSunAzimuth);

afb_ObjectReal_Out[2].tDataTimeOut := T#24H;
afb_ObjectReal_Out[2].eDataSource := _Domoticz_eDataSource.HTTP;
afb_ObjectReal_Out[2](scConnector := scConnector, 	uiIdentifier := uiIdentifier_SunAltitude,	rxUpdateInterlock := rxUpdateInterlock_int,			rValueAct => rSunAltitude);

afb_ObjectReal_Out[3].tDataTimeOut := T#24H;
afb_ObjectReal_Out[3].eDataSource := _Domoticz_eDataSource.HTTP;
afb_ObjectReal_Out[3](scConnector := scConnector, 	uiIdentifier := uiIdentifier_SunDistance,	rxUpdateInterlock := rxUpdateInterlock_int,			rValueAct => rSunDistance);

afb_ObjectReal_Out[4].tDataTimeOut := T#24H;
afb_ObjectReal_Out[4].eDataSource := _Domoticz_eDataSource.HTTP;
afb_ObjectReal_Out[4](scConnector := scConnector, 	uiIdentifier := uiIdentifier_MoonAzimuth,	rxUpdateInterlock := rxUpdateInterlock_int,			rValueAct => rMoonAzimuth);

afb_ObjectReal_Out[5].tDataTimeOut := T#24H;
afb_ObjectReal_Out[5].eDataSource := _Domoticz_eDataSource.HTTP;
afb_ObjectReal_Out[5](scConnector := scConnector, 	uiIdentifier := uiIdentifier_MoonAltitude,	rxUpdateInterlock := rxUpdateInterlock_int,			rValueAct => rMoonAltitude);

afb_ObjectReal_Out[6].tDataTimeOut := T#24H;
afb_ObjectReal_Out[6].eDataSource := _Domoticz_eDataSource.HTTP;
afb_ObjectReal_Out[6](scConnector := scConnector, 	uiIdentifier := uiIdentifier_MoonDistance,	rxUpdateInterlock := rxUpdateInterlock_int,			rValueAct => rMoonDistance);

afb_ObjectReal_Out[7].tDataTimeOut := T#24H;
afb_ObjectReal_Out[7].eDataSource := _Domoticz_eDataSource.HTTP;
afb_ObjectReal_Out[7](scConnector := scConnector, 	uiIdentifier := uiIdentifier_MoonPhase,		rxUpdateInterlock := rxUpdateInterlock_int,			rValueAct => rMoonPhase);

//Errors
fbEI_DataTimeOut.sInstanceName := sInstanceName;
fbEI_DataTimeOut.tErrorDelay := T#500MS;	//Give objects TIME TO be overruled BY other updates
fbEI_DataTimeOut(
	scConnector:= scConnector,
	xError:= xDataTimeOut_int
			AND (afb_ObjectReal_Out[1].xDataTimedOut
OR afb_ObjectReal_Out[2].xDataTimedOut
OR afb_ObjectReal_Out[3].xDataTimedOut
OR afb_ObjectReal_Out[4].xDataTimedOut
OR afb_ObjectReal_Out[5].xDataTimedOut
OR afb_ObjectReal_Out[6].xDataTimedOut
OR afb_ObjectReal_Out[7].xDataTimedOut),
	eErrorID:= Domoticz_eErrors.ObjectDataTimeOut
);
END_ACTION

END_FUNCTION_BLOCK

// Function Blocks/Hardware/Weather/Domoticz_WeatherBit
{attribute 'conditionalshow_all_locals'}
FUNCTION_BLOCK Domoticz_WeatherBit EXTENDS _Domoticz_Connector_Out
VAR_INPUT
	uiIdentifier_Temperature	:UINT;	//Temperature
	uiIdentifier_DewPoint		:UINT;	//Dew point
	uiIdentifier_Humidity		:UINT;	//Humidity
	uiIdentifier_Barometer		:UINT;	//Barometer
	uiIdentifier_Rain			:UINT;	//Rain rate and actual
	uiIdentifier_Wind			:UINT;	//Wind (direction,strenght)
	uiIdentifier_Visibility		:UINT;	//Visibility outside
	uiIdentifier_Cloudiness		:UINT;	//Cloudiness
	uiIdentifier_UV				:UINT;	//UV power
END_VAR
VAR_OUTPUT
	rTemperature				:REAL;
	rDewPoint					:REAL;
	rHumidity					:REAL;
	rBaroMeter					:REAL;
	rRain						:REAL;
	rRainRate					:REAL;
	rWindSpeed					:REAL;
	rWindGust					:REAL;
	rWindDirection				:REAL;
	rVisibility					:REAL;
	rCloudiness					:REAL;
	rUV							:REAL;
END_VAR
VAR
	afb_ObjectArrayReal_Out		:ARRAY[1..2] OF _Domoticz_ObjectArrayReal_Out;
	afb_ObjectReal_Out			:ARRAY[1..7] OF _Domoticz_ObjectReal_Out;
END_VAR

IF __ISVALIDREF(scConnector) THEN
	Main();
END_IF

ACTION Main:
{attribute 'conditionalshow'}
//Call parent function
SUPER^.Main();

//Set extended data timeout (Weather not updated frequently)
afb_ObjectArrayReal_Out[1].tDataTimeOut := T#24H;
afb_ObjectArrayReal_Out[2].tDataTimeOut := T#24H;
afb_ObjectReal_Out[1].tDataTimeOut := T#24H;
afb_ObjectReal_Out[2].tDataTimeOut := T#24H;
afb_ObjectReal_Out[3].tDataTimeOut := T#24H;
afb_ObjectReal_Out[4].tDataTimeOut := T#24H;
afb_ObjectReal_Out[5].tDataTimeOut := T#24H;
afb_ObjectReal_Out[6].tDataTimeOut := T#24H;
afb_ObjectReal_Out[7].tDataTimeOut := T#24H;

//Call all functions
//Extended data timeout (Weather not updated frequently)
afb_ObjectArrayReal_Out[1].tDataTimeOut := T#24H;
afb_ObjectArrayReal_Out[1].eDataSource := _Domoticz_eDataSource.HTTP;
afb_ObjectArrayReal_Out[1](	scConnector := scConnector, 	uiIdentifier := uiIdentifier_Wind,			rxUpdateInterlock := rxUpdateInterlock_int);

afb_ObjectArrayReal_Out[2].tDataTimeOut := T#24H;
afb_ObjectArrayReal_Out[2].eDataSource := _Domoticz_eDataSource.HTTP;
afb_ObjectArrayReal_Out[2](	scConnector := scConnector,		uiIdentifier := uiIdentifier_Rain,			rxUpdateInterlock := rxUpdateInterlock_int);
  
afb_ObjectReal_Out[1].tDataTimeOut := T#24H;
afb_ObjectReal_Out[1].eDataSource := _Domoticz_eDataSource.HTTP;                                                          
afb_ObjectReal_Out[1](		scConnector := scConnector, 	uiIdentifier := uiIdentifier_Temperature,	rxUpdateInterlock := rxUpdateInterlock_int,			rValueAct => rTemperature);

afb_ObjectReal_Out[2].tDataTimeOut := T#24H;
afb_ObjectReal_Out[2].eDataSource := _Domoticz_eDataSource.HTTP;
afb_ObjectReal_Out[2](		scConnector := scConnector, 	uiIdentifier := uiIdentifier_DewPoint,		rxUpdateInterlock := rxUpdateInterlock_int,			rValueAct => rDewPoint);

afb_ObjectReal_Out[3].tDataTimeOut := T#24H;
afb_ObjectReal_Out[3].eDataSource := _Domoticz_eDataSource.HTTP;
afb_ObjectReal_Out[3](		scConnector := scConnector, 	uiIdentifier := uiIdentifier_Humidity,		rxUpdateInterlock := rxUpdateInterlock_int,			rValueAct => rHumidity);

afb_ObjectReal_Out[4].tDataTimeOut := T#24H;
afb_ObjectReal_Out[4].eDataSource := _Domoticz_eDataSource.HTTP;
afb_ObjectReal_Out[4](		scConnector := scConnector, 	uiIdentifier := uiIdentifier_Barometer,		rxUpdateInterlock := rxUpdateInterlock_int,			rValueAct => rBaroMeter);

afb_ObjectReal_Out[5].tDataTimeOut := T#24H;
afb_ObjectReal_Out[5].eDataSource := _Domoticz_eDataSource.HTTP;
afb_ObjectReal_Out[5](		scConnector := scConnector, 	uiIdentifier := uiIdentifier_Visibility,	rxUpdateInterlock := rxUpdateInterlock_int,			rValueAct => rVisibility);

afb_ObjectReal_Out[6].tDataTimeOut := T#24H;
afb_ObjectReal_Out[6].eDataSource := _Domoticz_eDataSource.HTTP;
afb_ObjectReal_Out[6](		scConnector := scConnector, 	uiIdentifier := uiIdentifier_Cloudiness,	rxUpdateInterlock := rxUpdateInterlock_int,			rValueAct => rCloudiness);

afb_ObjectReal_Out[7].tDataTimeOut := T#24H;
afb_ObjectReal_Out[7].eDataSource := _Domoticz_eDataSource.HTTP;
afb_ObjectReal_Out[7](		scConnector := scConnector, 	uiIdentifier := uiIdentifier_UV,			rxUpdateInterlock := rxUpdateInterlock_int,			rValueAct => rUV);

//Output arrays
rWindSpeed	 	:= afb_ObjectArrayReal_Out[1].arValueAct[Domoticz_eSValues_Wind.Speed];
rWindGust		:= afb_ObjectArrayReal_Out[1].arValueAct[Domoticz_eSValues_Wind.Gust];
rWindDirection	:= afb_ObjectArrayReal_Out[1].arValueAct[Domoticz_eSValues_Wind.Bearing];

rRain		 	:= afb_ObjectArrayReal_Out[2].arValueAct[Domoticz_eSValues_Rain.Rain];
rRainRate		:= afb_ObjectArrayReal_Out[2].arValueAct[Domoticz_eSValues_Rain.RainRate];
											
//Errors
fbEI_DataTimeOut.sInstanceName := sInstanceName;
fbEI_DataTimeOut.tErrorDelay := T#500MS;	//Give objects TIME TO be overruled BY other updates
fbEI_DataTimeOut(
	scConnector:= scConnector,
	xError:= xDataTimeOut_int
			AND (afb_ObjectArrayReal_Out[1].xDataTimedOut
			OR afb_ObjectArrayReal_Out[2].xDataTimedOut
			OR afb_ObjectReal_Out[1].xDataTimedOut
			OR afb_ObjectReal_Out[2].xDataTimedOut
			OR afb_ObjectReal_Out[3].xDataTimedOut
			OR afb_ObjectReal_Out[4].xDataTimedOut
			OR afb_ObjectReal_Out[5].xDataTimedOut
			OR afb_ObjectReal_Out[6].xDataTimedOut
			OR afb_ObjectReal_Out[7].xDataTimedOut),
	eErrorID:= Domoticz_eErrors.ObjectDataTimeOut
);
END_ACTION

END_FUNCTION_BLOCK

// Functions/_Domoticz_StringToByte
{attribute 'conditionalshow_all_locals'}
{attribute 'conditionalshow'}
FUNCTION _Domoticz_StringToByte :BYTE
VAR_INPUT
	sData		:STRING(Domoticz_Constants.uiMaxSValuesize);	
END_VAR
VAR
END_VAR

//Extact data
IF sData = '1' OR sData = Domoticz_Constants.sData_On OR sData = Domoticz_Constants.sData_Open OR sData = Domoticz_Constants.sData_Locked OR sData = Domoticz_Constants.sData_Panic THEN
	_Domoticz_StringToByte := 1;
ELSIF sData = '0' OR sData = Domoticz_Constants.sData_Off OR sData = Domoticz_Constants.sData_Closed OR sData = Domoticz_Constants.sData_Unlocked OR sData = Domoticz_Constants.sData_Normal THEN
	_Domoticz_StringToByte := 0;
ELSE
	_Domoticz_StringToByte := 255;		//Invalid or unknown data
END_IF

END_FUNCTION

// Function Blocks/Server/_Domoticz_Server
{attribute 'conditionalshow_all_locals'}
{attribute 'conditionalshow'}
{attribute 'reflection'}
FUNCTION_BLOCK _Domoticz_Server EXTENDS _Domoticz_Connector
//VAR_IN_OUT
//	scConnector					:Domoticz_scServerSlaveConnector;
//END_VAR                     	
VAR_INPUT                   	
	//General               	
	xEnable						:BOOL;		//Enable FB
	xConnect					:BOOL;		//Connect to server(s)
END_VAR
VAR_OUTPUT
	//General
	scError						:Domoticz_scError;
	                        	
	//Output server status  	
	xConnected_HTTP				:BOOL;
	xConnected_MQTT				:BOOL;
	
END_VAR
VAR
	//{attribute 'instance-path'} 
	//{attribute 'noinit'}
	//sInstanceName 				:STRING(Domoticz_Constants.uiInstanceName);
	                        	
	//Parameters            	
	//Overall               	
	xAutoReconnect_int			:BOOL := TRUE;		//Auto reconnect after error
	                        	              
	//Data forcing          	
	tDataForceSetValues_int		:TIME := T#10S;		//Force set values if enabled after x time
	                        	
	//System time           	
	xAutoSyncClocks_int			:BOOL := TRUE;		//Sync system time with server
	tAutoSyncClocks_int			:TIME := T#3H;		//Time for each sync     
	                        	
	//Twilight              	
	todSunOffset_int			:TOD := TOD#00:30:00;	//Time offset (Pre-sunset) / (Post-sunrise)
	todSystemTime_Offset_int	:TOD := TOD#00:00:00;	//Time offset from server to show correct time on system
                            
	//HTTP                  
	sHTTP_IPAddress_int			:STRING(15) := '192.168.1.10';
	uiHTTP_ServerPort_int		:UINT := 8080;
	tHTTP_TimeOut_int			:TIME := T#3S;
	                        	
	//MQTT                  	
	sMQTT_IPAddress_int			:STRING(15) := '192.168.1.10';
	uiMQTT_ServerPort_int		:UINT := 1883;
	tMQTT_TimeOut_int			:TIME := T#3S;
	sMQTT_Username_int			:STRING(32);
	sMQTT_Password_int			:STRING(32);
	
	tMQTT_UpdateTimeOut_int		:TIME := T#60S;
	                        	
	//Internal          		
	wX, wY						:WORD;
	iCountMQTT_sValues			:INT;
	                        	
	TON_SlaveError_Reset		:TON;
	tSlaveErrorResetTime_int	:TIME := T#3S;
	ascActiveSlaveErrors_int	:ARRAY[1..Domoticz_Properties.uiActiveErrors] OF Domoticz_scError;
	
	psErrorInstance				:POINTER TO STRING(Domoticz_Constants.uiInstanceName);
	sErrorInstance_Concat		:STRING(Domoticz_Constants.uiInstanceName);
	psErrorInstance_Concat		:POINTER TO STRING(Domoticz_Constants.uiInstanceName);
                        	
	scError_Empty 				:Domoticz_scError;
	scObjectData_Empty			:Domoticz_scObjectData;

	//*************************************************************************************HTTP         	
	iStepper_HTTP				:INT;
	xConnected_HTTP_int			:BOOL;		//GET result was succesful > false on init/error state
	udiUpdateRate_HTTP_int		:UDINT;		//Internal counter
	udiUpdateRate_HTTP_mem		:UDINT;		//Internal counter
	uiObjectsPerConnection		:UDINT;		//scConnector.uiSlaveTotal/Domoticz_Properties.uiMaxHTTPConnections
	fbHTTP						:SNDLTN_HTTP.HTTP_Client;
	afbHTTP_Object				:ARRAY[1..Domoticz_Properties.uiMaxHTTPConnections] OF _Domoticz_Server_HTTP_Object;
	afbTON_ObjectExecute		:ARRAY[1..Domoticz_Properties.uiMaxHTTPConnections] OF TON;
	xHTTP_ObjectError			:BOOL;
	eHTTP_ObjectError			:Domoticz_eErrors;
	uiHTTP_ObjectError_wX		:UINT;
	uiHTTP_ObjectError_Source	:UINT;
	//
	TON_HTTP_UpdateServer		:TON;		//Update server values after set time
	//                      	
	xHTTP_StartUpDone			:BOOL;
	axHTTPStartUpDone			:ARRAY[1..Domoticz_Properties.uiMaxHTTPConnections] OF BOOL; //First reading done
	auiHTTPStartUpCycles		:ARRAY[1..Domoticz_Properties.uiMaxHTTPConnections] OF UINT; //First reading cycles done
	//                      	
	////Update of object    	
	auiHTTPUpdateIndex			:ARRAY[1..Domoticz_Properties.uiMaxHTTPConnections] OF UINT; //Index in array of server<>slave connetor
	xHTTP_NewObject				:BOOL;		//New object data available
	scHTTP_ObjectData_int		:Domoticz_scObjectData;		//Internal object data
	
	//Twilight time
	udiHTTP_Twilight			:UDINT;		//Epoch time
	
	//Used for concatting values
	sHTTP_Concat				:STRING(SNDLTN_HTTP.HTTP_Properties.uiHTTPMaxURLSize);
	psHTTP_Concat				:POINTER TO STRING(SNDLTN_HTTP.HTTP_Properties.uiHTTPMaxURLSize);
	sHTTP_ConcatHelper			:STRING(SNDLTN_HTTP.HTTP_Properties.uiHTTPMaxURLSize);
	psHTTP_ConcatHelper			:POINTER TO STRING(SNDLTN_HTTP.HTTP_Properties.uiHTTPMaxURLSize);
	                        	
	//JSON	                	
	fbHTTP_Parser				:SNDLTN_JSON.JSON_Parser;
	fbHTTP_Values				:SNDLTN_JSON.JSON_GetMultiValue;
	                        	
	TON_HTTP_UpdateTimeOut		:TON;
	//*************************************************************************************MQTT
	iStepper_MQTT				:INT;
	xConnected_MQTT_int			:BOOL;		//Output of MQTT FB
	udiUpdateRate_MQTT_int		:UDINT;		//Internal counter
	udiUpdateRate_MQTT_mem		:UDINT;		//Internal counter
	fbMQTT_Receive				:SNDLTN_MQTT.MQTT_Client;
	fbMQTT_Send					:SNDLTN_MQTT.MQTT_Client;
	                        	
	//Update of object      	
	xMQTT_NewObject				:BOOL;		//New object data available
	scMQTT_ObjectData_int		:Domoticz_scObjectData;		//Internal object data
                            	
	//Output                	
	rMQTT_ColorTemperature		:REAL;		//Calculation helper
	TON_MQTT_PublishTimeout		:TON;		//Timeout publishing
	
	//Used for concatting values
	sMQTT_Concat				:STRING(SNDLTN_MQTT.MQTT_Properties.uiMQTTMaxMessageSize);
	psMQTT_Concat				:POINTER TO STRING(SNDLTN_MQTT.MQTT_Properties.uiMQTTMaxMessageSize);
	sMQTT_ConcatHelper			:STRING(SNDLTN_MQTT.MQTT_Properties.uiMQTTMaxMessageSize);
	psMQTT_ConcatHelper			:POINTER TO STRING(SNDLTN_MQTT.MQTT_Properties.uiMQTTMaxMessageSize);
		                    		
	//JSON	                	
	fbMQTT_Parser				:SNDLTN_JSON.JSON_Parser;
	fbMQTT_Values				:SNDLTN_JSON.JSON_GetMultiValue;
	                        	
	TON_MQTT_UpdateTimeOut		:TON;
	
	//*************************************************************************************TIME
	//System time
	FB_SysTime_Get				:RTCLK.GetDateAndTime;
	FB_SysTime_Set				:RTCLK.SetDateAndTime;
	udiSysTime_Set				:UDINT;	
	TP_SysTime					:TP;		//Cycle read time
	xSyncTime_int				:BOOL;		//Sync time command from HTTP
	                        	
	scTwilightData_Empty		:Domoticz_scTwilightData;
END_VAR

Main();

ACTION Main:
{attribute 'conditionalshow'}
//Call parent function
SUPER^.Main();

{warning disable C0139}
//Resolve SA0033 error by calling values
Domoticz_Constants.uiObjectData_Type; 
Domoticz_Constants.uiErrorInfoSize;
{warning restore C0139}

IF xEnable THEN
	//Call actions
	MQTT_Main();			//Start MQTT
	HTTP_Main();			//Start HTTP
	
	//Distribute update if available
	IF scConnector.xNewObject_Rx THEN
		scConnector.xNewObject_Rx := FALSE;
		scConnector.scObjectData_Rx := scObjectData_Empty;
	ELSIF xMQTT_NewObject AND NOT scConnector.xNewObject_Rx THEN
		scConnector.scObjectData_Rx := scMQTT_ObjectData_int;
		xMQTT_NewObject := FALSE;
		scConnector.xNewObject_Rx := TRUE;
	ELSIF xHTTP_NewObject AND NOT scConnector.xNewObject_Rx THEN
		scConnector.scObjectData_Rx := scHTTP_ObjectData_int;
		xHTTP_NewObject := FALSE;
		scConnector.xNewObject_Rx := TRUE;
	END_IF
	
	//Update system time
	SystemTime();
	
	
	//OUTPUTS
		
	//Data forcing
	scConnector.tDataForceSetValues := tDataForceSetValues_int;
	
	//Server status
	scConnector.xServerConnected := xHTTP_StartUpDone
									AND xConnected_HTTP_int 	
									AND xConnected_MQTT_int;
	
	//Set data source from PLC
	scConnector.scObjectData_TX.eSource := _Domoticz_eDataSource.PLC;	
	
	//Refresh / recount total registered slaves
	scConnector.uiSlaveTotal := 0;
	FOR wX := 1 TO Domoticz_Properties.uiMaxConnectedSlaves DO
		IF scConnector.auiSlaveIdentifier[wX] > 0 THEN
			scConnector.uiSlaveTotal := scConnector.uiSlaveTotal + 1;
		END_IF
	END_FOR
	
	//Call error handling
	ErrorHandling();
		
	//Outputs
	xConnected_HTTP := xConnected_HTTP_int;
	TON_HTTP_UpdateTimeOut(IN:=udiUpdateRate_HTTP_mem=udiUpdateRate_HTTP_int,PT:=tHTTP_TimeOut_int);	//Guard update rate
	IF udiUpdateRate_HTTP_mem <> udiUpdateRate_HTTP_int THEN udiUpdateRate_HTTP_mem := udiUpdateRate_HTTP_int; END_IF

	xConnected_MQTT := xConnected_MQTT_int;
	TON_MQTT_UpdateTimeOut(IN:=udiUpdateRate_MQTT_mem=udiUpdateRate_MQTT_int,PT:=tMQTT_UpdateTimeOut_int);	//Guard update rate
	IF udiUpdateRate_MQTT_mem <> udiUpdateRate_MQTT_int THEN udiUpdateRate_MQTT_mem := udiUpdateRate_MQTT_int; END_IF
	
//Reset all outputs when disabled
ELSE 
	scError.xError 							:= FALSE;
	scError.eErrorID 						:= Domoticz_eErrors.NoError;
	
	scError.sErrorInfo							:= '';
	scError.sErrorInstance							:= '';
	xConnected_HTTP_int						:= FALSE;
	xConnected_MQTT_int						:= FALSE;
	xConnected_HTTP							:= FALSE;
	xConnected_MQTT							:= FALSE;
	FOR wX := 1 TO Domoticz_Properties.uiMaxConnectedSlaves DO
		scConnector.auiSlaveIdentifier[wX]	:= 0;
	END_FOR
	scConnector.uiSlaveTotal				:= 0;
	scConnector.scTwilightData				:= scTwilightData_Empty;
	scConnector.xNewObject_Tx				:= FALSE;
	scConnector.scObjectData_Tx				:= scObjectData_Empty;
	scConnector.xNewObject_Rx				:= FALSE;
	scConnector.scObjectData_Rx				:= scObjectData_Empty;
	scConnector.xServerConnected			:= FALSE;
	scConnector.scSlaveError.xError			:= FALSE;
	scConnector.scSlaveError.eErrorID 		:= Domoticz_eErrors.NoError;
	scConnector.scSlaveError.sErrorInstance := '';
	scConnector.scSlaveError.sErrorInfo 	:= '';
	scConnector.tDataForceSetValues			:= T#5S;
	udiUpdateRate_HTTP_int					:= 0;
	udiUpdateRate_MQTT_int					:= 0;
END_IF
END_ACTION

{attribute 'monitoring' := 'call'} PROPERTY udiUpdateRate_HTTP :UDINT
GET
udiUpdateRate_HTTP := udiUpdateRate_HTTP_int;
END_GET
END_PROPERTY

ACTION HTTP_DataTwilight:
{attribute 'conditionalshow'}

//HTTP

//Get pointers
psHTTP_Concat := ADR(sHTTP_Concat);
psHTTP_ConcatHelper := ADR(sHTTP_ConcatHelper);

//Construct URL

//HTTP://
sHTTP_Concat := Domoticz_Constants.sURL_HTTP;

//Add server IP
StrConcatA(ADR(sHTTP_IPAddress_int), psHTTP_Concat, TO_INT(SNDLTN_HTTP.HTTP_Properties.uiHTTPMaxURLSize));

//Add seperator
sHTTP_ConcatHelper := ':';
StrConcatA(psHTTP_ConcatHelper, psHTTP_Concat, TO_INT(SNDLTN_HTTP.HTTP_Properties.uiHTTPMaxURLSize));

//Add server port
sHTTP_ConcatHelper := TO_STRING(uiHTTP_ServerPort_int);
StrConcatA(psHTTP_ConcatHelper, psHTTP_Concat, TO_INT(SNDLTN_HTTP.HTTP_Properties.uiHTTPMaxURLSize));

//Add request
StrConcatA(ADR(Domoticz_Constants.sURL_Twilight), psHTTP_Concat, TO_INT(SNDLTN_HTTP.HTTP_Properties.uiHTTPMaxURLSize));

//Get data from HTTP/JSON
fbHTTP.sURL := sHTTP_Concat;
fbHTTP.eRequestType := HTTP_eRequestType.GET;

//Specify data

//Server name
fbHTTP_Values.asPropertyName[1] 		:= Domoticz_Constants.sPropertyHTTP_AstronomicRise;
fbHTTP_Values.aeConversionType[1] 		:= JSON_eConversionType.TimeOfDay;
                                    	
//Update URL                        	
fbHTTP_Values.asPropertyName[2] 		:= Domoticz_Constants.sPropertyHTTP_AstronomicSet;
fbHTTP_Values.aeConversionType[2] 		:= JSON_eConversionType.TimeOfDay;
                                    	
//nValue                            	
fbHTTP_Values.asPropertyName[3] 		:= Domoticz_Constants.sPropertyHTTP_CivilRise;
fbHTTP_Values.aeConversionType[3] 		:= JSON_eConversionType.TimeOfDay;
                                    	
//sValue1                           	
fbHTTP_Values.asPropertyName[4] 		:= Domoticz_Constants.sPropertyHTTP_CivilSet;
fbHTTP_Values.aeConversionType[4] 		:= JSON_eConversionType.TimeOfDay;
                                    	
//sValue2                           	
fbHTTP_Values.asPropertyName[5] 		:= Domoticz_Constants.sPropertyHTTP_NauticRise;
fbHTTP_Values.aeConversionType[5] 		:= JSON_eConversionType.TimeOfDay;
                                    	
//sValue3                           	
fbHTTP_Values.asPropertyName[6] 		:= Domoticz_Constants.sPropertyHTTP_NauticSet;
fbHTTP_Values.aeConversionType[6] 		:= JSON_eConversionType.TimeOfDay;
                                    	
//sValue4                           	
fbHTTP_Values.asPropertyName[7] 		:= Domoticz_Constants.sPropertyHTTP_SunRise;
fbHTTP_Values.aeConversionType[7] 		:= JSON_eConversionType.TimeOfDay;
                                    	
//sValue5                           	
fbHTTP_Values.asPropertyName[8] 		:= Domoticz_Constants.sPropertyHTTP_SunSet;
fbHTTP_Values.aeConversionType[8] 		:= JSON_eConversionType.TimeOfDay;
                                    	
//sValue5                           	
fbHTTP_Values.asPropertyName[9] 		:= Domoticz_Constants.sPropertyHTTP_AtSouth;
fbHTTP_Values.aeConversionType[9] 		:= JSON_eConversionType.TimeOfDay;
                                    	
//sValue5                           	
fbHTTP_Values.asPropertyName[10] 		:= Domoticz_Constants.sPropertyHTTP_DayLength;
fbHTTP_Values.aeConversionType[10] 	:= JSON_eConversionType.TimeOfDay;
                                    	
//sValue5                           	
fbHTTP_Values.asPropertyName[11] 		:= Domoticz_Constants.sPropertyHTTP_SystemTime;
fbHTTP_Values.aeConversionType[11] 	:= JSON_eConversionType.DateAndTime;

//Disable all other conversions
FOR wX := 12 TO SNDLTN_JSON.JSON_Properties.uiJSONMaxInputMultiValue DO 
	fbHTTP_Values.asPropertyName[wX]	:= '';
	fbHTTP_Values.aeConversionType[wX]:= JSON_eConversionType.None; 
END_FOR	

//******************************************************************JSON:PARSE
IF fbHTTP.xDone AND fbHTTP.xResponseValid THEN
		
	IF fbHTTP_Values.axMatchFound[1] THEN	
		scConnector.scTwilightData.todAstronomicRise := fbHTTP_Values.atodPropertyValue[1];
	ELSE
		scConnector.scTwilightData.todAstronomicRise := TOD#0:0:0;
	END_IF
	
	IF fbHTTP_Values.axMatchFound[2] THEN
		scConnector.scTwilightData.todAstronomicSet := fbHTTP_Values.atodPropertyValue[2];
	ELSE
		scConnector.scTwilightData.todAstronomicSet := TOD#0:0:0;
	END_IF
	
	IF fbHTTP_Values.axMatchFound[3] THEN
		scConnector.scTwilightData.todCivilRise := fbHTTP_Values.atodPropertyValue[3];
	ELSE
		scConnector.scTwilightData.todCivilRise := TOD#0:0:0;
	END_IF
	
	IF fbHTTP_Values.axMatchFound[4] THEN
		scConnector.scTwilightData.todCivilSet := fbHTTP_Values.atodPropertyValue[4];
	ELSE
		scConnector.scTwilightData.todCivilSet := TOD#0:0:0;
	END_IF
	
	IF fbHTTP_Values.axMatchFound[5] THEN
		scConnector.scTwilightData.todNauticRise := fbHTTP_Values.atodPropertyValue[5];
	ELSE
		scConnector.scTwilightData.todNauticRise := TOD#0:0:0;
	END_IF
	
	IF fbHTTP_Values.axMatchFound[6] THEN
		scConnector.scTwilightData.todNauticSet := fbHTTP_Values.atodPropertyValue[6];
	ELSE
		scConnector.scTwilightData.todNauticSet := TOD#0:0:0;
	END_IF
	
	IF fbHTTP_Values.axMatchFound[7] THEN
		//Sunrise
		scConnector.scTwilightData.todSunRise := fbHTTP_Values.atodPropertyValue[7];
		
		//Pre-sunrise
		udiHTTP_Twilight := TO_UDINT(scConnector.scTwilightData.todSunRise) - TO_UDINT(todSunOffset_int);
		scConnector.scTwilightData.todPreSunRise := TO_TOD(udiHTTP_Twilight);
		
		//Post-sunrise
		udiHTTP_Twilight := TO_UDINT(scConnector.scTwilightData.todSunRise) + TO_UDINT(todSunOffset_int);
		scConnector.scTwilightData.todPostSunRise := TO_TOD(udiHTTP_Twilight);
	ELSE
		scConnector.scTwilightData.todPreSunRise := TOD#0:0:0;
		scConnector.scTwilightData.todSunRise := TOD#0:0:0;
		scConnector.scTwilightData.todPostSunRise := TOD#0:0:0;
	END_IF
	
	IF fbHTTP_Values.axMatchFound[8] THEN
		//Sunset
		scConnector.scTwilightData.todSunSet := fbHTTP_Values.atodPropertyValue[8];
		
		//Pre-sunset
		udiHTTP_Twilight := TO_UDINT(scConnector.scTwilightData.todSunSet) - TO_UDINT(todSunOffset_int);
		scConnector.scTwilightData.todPreSunSet := TO_TOD(udiHTTP_Twilight);
		
		//Post-sunset
		udiHTTP_Twilight := TO_UDINT(scConnector.scTwilightData.todSunSet) + TO_UDINT(todSunOffset_int);
		scConnector.scTwilightData.todPostSunSet := TO_TOD(udiHTTP_Twilight);
	ELSE
		scConnector.scTwilightData.todPreSunSet := TOD#0:0:0;
		scConnector.scTwilightData.todSunSet := TOD#0:0:0;
		scConnector.scTwilightData.todPostSunSet := TOD#0:0:0;
	END_IF
	
	IF fbHTTP_Values.axMatchFound[9] THEN
		scConnector.scTwilightData.todSunAtSouth := fbHTTP_Values.atodPropertyValue[9];
	ELSE
		scConnector.scTwilightData.todSunAtSouth := TOD#0:0:0;
	END_IF
	
	IF fbHTTP_Values.axMatchFound[10] THEN
		scConnector.scTwilightData.todDayLength := fbHTTP_Values.atodPropertyValue[10];
	ELSE
		scConnector.scTwilightData.todDayLength := TOD#0:0:0;
	END_IF
	
	IF fbHTTP_Values.axMatchFound[11] THEN
		scConnector.scTwilightData.dtServer := fbHTTP_Values.adtPropertyValue[11];
	ELSE
		scConnector.scTwilightData.dtServer := DT#1970-1-1-0:0:0;
	END_IF
END_IF
END_ACTION

ACTION MQTT_Main:
{attribute 'conditionalshow'}

CASE iStepper_MQTT OF

	-10:	//Error
	//Reset if needed
	IF NOT xConnect OR xAutoReconnect_int THEN
		fbMQTT_Parser.xResetError := TRUE;
		iStepper_MQTT := 0;
	END_IF
	
	0:	//Disabled
	fbMQTT_Receive.xConnect := FALSE;
	fbMQTT_Receive.xSubscribe := FALSE;
	fbMQTT_Send.xConnect := FALSE;
	fbMQTT_Send.xSubscribe := FALSE;
	
	fbMQTT_Parser.xResetError := FALSE;
	
	scConnector.xNewObject_Tx := FALSE;	//Revoke send command busy
	
	//Wait for connect command
	IF xConnect THEN
		iStepper_MQTT := 10;
	END_IF
	
	10:	//Connect MQTT function block
	fbMQTT_Receive.xConnect := TRUE;
	fbMQTT_Send.xConnect := TRUE;
	
	//Wait for connection done
	IF fbMQTT_Receive.xConnected AND fbMQTT_Send.xConnected THEN
		iStepper_MQTT := 20;
	//Error occured (outputted in main)
	ELSIF fbMQTT_Receive.xError OR fbMQTT_Send.xError THEN
		iStepper_MQTT := -10;
	END_IF
	
	20:	//Subscribe to out topic
	fbMQTT_Receive.xSubscribe := TRUE;
	//Sending topic doesn't subscribe to anything
	//Wait for connection done
	IF fbMQTT_Receive.xSubscribed THEN
		iStepper_MQTT := 30;
	//Error occured (outputted in main)
	ELSIF fbMQTT_Receive.xError OR fbMQTT_Send.xError THEN
		iStepper_MQTT := -10;
	END_IF
	
	30:	//Ready
	
	//Process incoming data
	MQTT_DataObject_In();
	
	//Process outgoing data
	MQTT_DataObject_Out ();	//Build message

	//Wait for user to break connection
	IF NOT xConnect THEN
		iStepper_MQTT := 0;
	//Error occured (outputted in main)
	ELSIF fbMQTT_Receive.xError OR fbMQTT_Send.xError OR fbMQTT_Parser.xError THEN
		iStepper_MQTT := -10;
	END_IF

END_CASE

fbMQTT_Receive(
	xEnable:= TRUE, 
	xConnect:= , 
	tTimeOut:= tMQTT_TimeOut_int, 
	sBrokerIP:= sMQTT_IPAddress_int, 
	uiBrokerPort:= uiMQTT_ServerPort_int, 
	sBrokerUser:= sMQTT_Username_int, 
	sBrokerPass:= sMQTT_Password_int, 
	xSubscribe:= , 
	sSubscribeTopic:= Domoticz_Properties.sMQTT_TopicReceive, 
	xPublish:= , 
	sPublishTopic:= , 
	sPublishMessage:= , 
	xPublishRetain:= , 
	sLastWillTopic:= , 
	sLastWillMessage:= , 
	xLastWillRetain:= , 
	eState=> , 
	xError=> , 
	eErrorID=> , 
	xConnected=> , 
	xSubscribed=> , 
	xPublished=> , 
	xSubscriptionNewMessage=> , 
	sSubscriptionTopic=> , 
	sSubscriptionMessage=>  
);

fbMQTT_Send(
	xEnable:= TRUE, 
	xConnect:= , 
	tTimeOut:= tMQTT_TimeOut_int, 
	sBrokerIP:= sMQTT_IPAddress_int, 
	uiBrokerPort:= uiMQTT_ServerPort_int, 
	sBrokerUser:= sMQTT_Username_int, 
	sBrokerPass:= sMQTT_Password_int, 
	xSubscribe:= , 
	sSubscribeTopic:= , 
	xPublish:= , 
	sPublishTopic:= Domoticz_Properties.sMQTT_TopicSend, 
	sPublishMessage:= , 
	xPublishRetain:= , 
	sLastWillTopic:= , 
	sLastWillMessage:= , 
	xLastWillRetain:= , 
	eState=> , 
	xError=> , 
	eErrorID=> , 
	xConnected=> , 
	xSubscribed=> , 
	xPublished=> , 
	xSubscriptionNewMessage=> , 
	sSubscriptionTopic=> , 
	sSubscriptionMessage=> 
);

xConnected_MQTT_int := fbMQTT_Receive.xConnected AND fbMQTT_Send.xConnected;

//Parse MQTT message > only processed if input changes	
fbMQTT_Parser(
	xResetError:= , 
	sContent:= fbMQTT_Receive.sSubscriptionMessage, 
);
	
fbMQTT_Values(
	pasProperties:= ADR(fbMQTT_Parser.asProperties[0,0]), 
	asPropertyName:= , 
	aeConversionType:= , 
);
	
//Reset statistics
IF NOT fbMQTT_Receive.xConnected OR NOT fbMQTT_Send.xConnected THEN
	udiUpdateRate_MQTT_int := 0;
END_IF
END_ACTION

ACTION HTTP_Main:
{attribute 'conditionalshow'}
//Twilight update > also used for connection check
CASE iStepper_HTTP OF

	-10:	//Error
	xConnected_HTTP_int := FALSE;			//Set output status
	
	//Reset if needed
	IF NOT xConnect OR xAutoReconnect_int THEN
		fbHTTP_Parser.xResetError := TRUE;
		iStepper_HTTP := 0;
	END_IF
	
	0:	//Disabled
	
	fbHTTP.xExecute := FALSE;
	fbHTTP_Parser.xResetError := FALSE;
	
	//Reset
	FOR wX := 1 TO Domoticz_Properties.uiMaxHTTPConnections DO
		auiHTTPStartUpCycles[wX] := 0;
		axHTTPStartUpDone[wX] := FALSE;
	END_FOR
	
	//Wait for connect command
	IF xConnect THEN
		iStepper_HTTP := 10;
	ELSE
		xConnected_HTTP_int := FALSE;			//Set output status
	END_IF
	
	10:	//Get twilight data
	
	//Reset timer
	TON_HTTP_UpdateServer(IN:=FALSE);
	
	HTTP_DataTwilight();	//Process data
	
	fbHTTP.xExecute := TRUE;
	
	//Wait for done
	//Not all data received, retrigger
	IF fbHTTP.xDone AND NOT fbHTTP.xResponseValid THEN
		fbHTTP.xExecute := FALSE;
	//All data received, continue
	ELSIF fbHTTP.xDone AND fbHTTP.xResponseValid  THEN
		xConnected_HTTP_int := TRUE;	//Set output status
		fbHTTP.xExecute := FALSE;
		udiUpdateRate_HTTP_int := udiUpdateRate_HTTP_int + 1;	//Update statistics
		xSyncTime_int := TRUE;	//Update local time
		iStepper_HTTP := 20;
	//Error occured (outputted in main)
	ELSIF fbHTTP.xError OR fbHTTP_Parser.xError THEN
		iStepper_HTTP := -10;
	END_IF
	
	20:	//Ready
	
	//Run timer to update server values	
	TON_HTTP_UpdateServer(IN:=TRUE, PT:=tAutoSyncClocks_int);
	
	//Wait for user to break connection
	IF NOT xConnect THEN 
		iStepper_HTTP := 0;
	//Run Twilight update
	ELSIF TON_HTTP_UpdateServer.Q THEN
		iStepper_HTTP := 10;
	//Error occured (outputted in main)
	ELSIF fbHTTP.xError OR fbHTTP_Parser.xError THEN
		iStepper_HTTP := -10;
	END_IF
	
END_CASE

//Reset data before FOR-loop
xHTTP_ObjectError := FALSE;
eHTTP_ObjectError := Domoticz_eErrors.NoError;
uiHTTP_ObjectError_wX := 0;
uiHTTP_ObjectError_Source := 0;
xHTTP_StartUpDone := TRUE;

uiObjectsPerConnection := TO_UINT(scConnector.uiSlaveTotal/Domoticz_Properties.uiMaxHTTPConnections) + 1 + 1;	//Compensate for value after decimals and for array start at zero

FOR wX := 1 TO (Domoticz_Properties.uiMaxHTTPConnections) DO
	//Run timer, give other elements time to publish data
	afbTON_ObjectExecute[wX](IN:= , PT:= T#100MS, Q=> , ET=> );	

	//Functions
	afbHTTP_Object[wX](
		sIPAddress:= sHTTP_IPAddress_int, 
		uiServerPort:= uiHTTP_ServerPort_int, 
		tTimeOut:= tHTTP_TimeOut_int, 
		dtTimeStamp:= scConnector.scTwilightData.dtSystem, 
		xReadData:= afbTON_ObjectExecute[wX].Q, 
		//									//Array starts at 1 	//Identifiers	//FB Number offset minus 1
		uiIdentifier:= scConnector.auiSlaveIdentifier[1 + auiHTTPUpdateIndex[wX] + ((wX-1) * uiObjectsPerConnection)], 
		xError=> , 
		xBusy=> , 
		xDone=> , 
		scObjectData=> );
		
	//Check if error active
	IF afbHTTP_Object[wX].xError
	AND afbHTTP_Object[wX].eErrorID <> Domoticz_eErrors.HTTP_InvalidIdentifier THEN 	//Ignore identifier 0
		xHTTP_ObjectError := TRUE;
		eHTTP_ObjectError := afbHTTP_Object[wX].eErrorID;
		uiHTTP_ObjectError_wX := afbHTTP_Object[wX].uiIdentifier;
		uiHTTP_ObjectError_Source := wX;
	END_IF
	
	//Check if first startup done or not
	IF NOT axHTTPStartUpDone[wX] THEN xHTTP_StartUpDone := FALSE; END_IF
		
	//Activate reading (one-cycle low)
	IF NOT afbTON_ObjectExecute[wX].IN THEN afbTON_ObjectExecute[wX].IN := TRUE; END_IF
		
	//Wait until function done
	IF afbHTTP_Object[wX].xDone AND NOT xHTTP_NewObject
	OR afbHTTP_Object[wX].xError THEN
		//Only publish when done
		IF afbHTTP_Object[wX].xDone THEN
			//Publish info
			scHTTP_ObjectData_int := afbHTTP_Object[wX].scObjectData;
			xHTTP_NewObject := TRUE;	
			udiUpdateRate_HTTP_int := udiUpdateRate_HTTP_int+1;
		END_IF
		//Reset
		afbTON_ObjectExecute[wX].IN := FALSE;
		//Increase index
		IF auiHTTPUpdateIndex[wX] < uiObjectsPerConnection THEN
			auiHTTPUpdateIndex[wX] := auiHTTPUpdateIndex[wX] + 1;
		//List done, restart list
		ELSE
			auiHTTPUpdateIndex[wX] := 0;
			//Count startup cycles
			IF auiHTTPStartUpCycles[wX] < Domoticz_Properties.uiHTTPStartUpCycles THEN
				auiHTTPStartUpCycles[wX] := auiHTTPStartUpCycles[wX] + 1;
			//Startup done
			ELSE
				axHTTPStartUpDone[wX] := TRUE;
			END_IF
		END_IF
	END_IF
END_FOR

//HTTP Server
fbHTTP(
	xExecute:= , 
	udiTimeOut:= TIME_TO_UDINT(tHTTP_TimeOut_int)*1000, 
);

//Parse HTTP content > only processed if input changes
fbHTTP_Parser(
	xResetError:= , 
	sContent:= fbHTTP.scResponse.sContent, 
);
	
//Get JSON values
fbHTTP_Values(
	pasProperties:= ADR(fbHTTP_Parser.asProperties[0,0]), 
	asPropertyName:= , 
	aeConversionType:= , 
);

//Reset statistics
IF NOT xConnected_HTTP_int THEN
	udiUpdateRate_HTTP_int := 0;
END_IF
END_ACTION

ACTION MQTT_DataObject_In:
{attribute 'conditionalshow'}

//MQTT

//Specify data

//Identifier
fbMQTT_Values.asPropertyName[_Domoticz_eMQTT_PropertyNames.Identifier] 		:= Domoticz_Constants.sPropertyMQTT_idx;
fbMQTT_Values.aeConversionType[_Domoticz_eMQTT_PropertyNames.Identifier] 	:= JSON_eConversionType.UnsignedInteger;
      
//Object Type                              	
fbMQTT_Values.asPropertyName[_Domoticz_eMQTT_PropertyNames.ObjectType] 		:= Domoticz_Constants.sPropertyMQTT_DType;
fbMQTT_Values.aeConversionType[_Domoticz_eMQTT_PropertyNames.ObjectType] 	:= JSON_eConversionType.None;
                              	
//Switch Type                              	
fbMQTT_Values.asPropertyName[_Domoticz_eMQTT_PropertyNames.SwitchType] 		:= Domoticz_Constants.sPropertyMQTT_SType;
fbMQTT_Values.aeConversionType[_Domoticz_eMQTT_PropertyNames.SwitchType] 	:= JSON_eConversionType.None;
                                    	
//nValue                            	
fbMQTT_Values.asPropertyName[_Domoticz_eMQTT_PropertyNames.NValue] 			:= Domoticz_Constants.sPropertyMQTT_NValue;
fbMQTT_Values.aeConversionType[_Domoticz_eMQTT_PropertyNames.NValue] 		:= JSON_eConversionType.Integer;
                                    	
//sValue1                           	
fbMQTT_Values.asPropertyName[_Domoticz_eMQTT_PropertyNames.SValue1] 		:= Domoticz_Constants.sPropertyMQTT_SValue1;
fbMQTT_Values.aeConversionType[_Domoticz_eMQTT_PropertyNames.SValue1] 		:= JSON_eConversionType.None;
                                    	
//sValue2                           	
fbMQTT_Values.asPropertyName[_Domoticz_eMQTT_PropertyNames.SValue2] 		:= Domoticz_Constants.sPropertyMQTT_SValue2;
fbMQTT_Values.aeConversionType[_Domoticz_eMQTT_PropertyNames.SValue2] 		:= JSON_eConversionType.None;
                                    	
//sValue3                           	
fbMQTT_Values.asPropertyName[_Domoticz_eMQTT_PropertyNames.SValue3] 		:= Domoticz_Constants.sPropertyMQTT_SValue3;
fbMQTT_Values.aeConversionType[_Domoticz_eMQTT_PropertyNames.SValue3] 		:= JSON_eConversionType.None;
                                    	
//sValue4                           	
fbMQTT_Values.asPropertyName[_Domoticz_eMQTT_PropertyNames.SValue4] 		:= Domoticz_Constants.sPropertyMQTT_SValue4;
fbMQTT_Values.aeConversionType[_Domoticz_eMQTT_PropertyNames.SValue4] 		:= JSON_eConversionType.None;
                                    	
//sValue5                           	
fbMQTT_Values.asPropertyName[_Domoticz_eMQTT_PropertyNames.SValue5] 		:= Domoticz_Constants.sPropertyMQTT_SValue5;
fbMQTT_Values.aeConversionType[_Domoticz_eMQTT_PropertyNames.SValue5] 		:= JSON_eConversionType.None;

//sValue6                       	
fbMQTT_Values.asPropertyName[_Domoticz_eMQTT_PropertyNames.SValue6] 		:= Domoticz_Constants.sPropertyMQTT_SValue6;
fbMQTT_Values.aeConversionType[_Domoticz_eMQTT_PropertyNames.SValue6] 		:= JSON_eConversionType.None;

//Color (R)                         	
fbMQTT_Values.asPropertyName[_Domoticz_eMQTT_PropertyNames.ColorR] 			:= Domoticz_Constants.asProperty_Colors[Domoticz_eSValues_Colors.Red];
fbMQTT_Values.aeConversionType[_Domoticz_eMQTT_PropertyNames.ColorR] 		:= JSON_eConversionType.None;
//Color (G)                         	
fbMQTT_Values.asPropertyName[_Domoticz_eMQTT_PropertyNames.ColorG] 			:= Domoticz_Constants.asProperty_Colors[Domoticz_eSValues_Colors.Green];
fbMQTT_Values.aeConversionType[_Domoticz_eMQTT_PropertyNames.ColorG] 		:= JSON_eConversionType.None;
//Color (B)                           	
fbMQTT_Values.asPropertyName[_Domoticz_eMQTT_PropertyNames.ColorB] 			:= Domoticz_Constants.asProperty_Colors[Domoticz_eSValues_Colors.Blue];
fbMQTT_Values.aeConversionType[_Domoticz_eMQTT_PropertyNames.ColorB] 		:= JSON_eConversionType.None;
//Color (CW)                          	
fbMQTT_Values.asPropertyName[_Domoticz_eMQTT_PropertyNames.ColorCW] 		:= Domoticz_Constants.asProperty_Colors[Domoticz_eSValues_Colors.ColdWhite];
fbMQTT_Values.aeConversionType[_Domoticz_eMQTT_PropertyNames.ColorCW] 		:= JSON_eConversionType.None;
//Color (WW)                            	
fbMQTT_Values.asPropertyName[_Domoticz_eMQTT_PropertyNames.ColorWW] 		:= Domoticz_Constants.asProperty_Colors[Domoticz_eSValues_Colors.WarmWhite];
fbMQTT_Values.aeConversionType[_Domoticz_eMQTT_PropertyNames.ColorWW] 		:= JSON_eConversionType.None;

//Reset data on start
IF NOT fbMQTT_Receive.xSubscriptionNewMessage
AND NOT xMQTT_NewObject THEN
	FOR wX := 1 TO Domoticz_Constants.uiMaxSValues DO
		scMQTT_ObjectData_int.asValue[wX] := '';
	END_FOR		
END_IF

//*****************************************************************************************************		
//Set all data if input changed (see below)
IF fbMQTT_Receive.xSubscriptionNewMessage THEN
	
	//Identifier
	IF fbMQTT_Values.axMatchFound[_Domoticz_eMQTT_PropertyNames.Identifier] THEN
		scMQTT_ObjectData_int.uiIdentifier := fbMQTT_Values.auiPropertyValue[_Domoticz_eMQTT_PropertyNames.Identifier];
	ELSE
		scMQTT_ObjectData_int.uiIdentifier := 0;
	END_IF
	
	//nValue
	IF fbMQTT_Values.axMatchFound[_Domoticz_eMQTT_PropertyNames.NValue] THEN
		scMQTT_ObjectData_int.iValue := fbMQTT_Values.aiPropertyValue[_Domoticz_eMQTT_PropertyNames.NValue];
	ELSE
		scMQTT_ObjectData_int.iValue := 0;
	END_IF
	
	//sValue1	
	IF fbMQTT_Values.axMatchFound[_Domoticz_eMQTT_PropertyNames.SValue1] THEN
		scMQTT_ObjectData_int.asValue[1] := fbMQTT_Values.asPropertyValue[_Domoticz_eMQTT_PropertyNames.SValue1];
	ELSE
		scMQTT_ObjectData_int.asValue[1] := '';
	END_IF
    
	//sValue2	
	IF fbMQTT_Values.axMatchFound[_Domoticz_eMQTT_PropertyNames.SValue2] THEN
		scMQTT_ObjectData_int.asValue[2] := fbMQTT_Values.asPropertyValue[_Domoticz_eMQTT_PropertyNames.SValue2];
	ELSE
		scMQTT_ObjectData_int.asValue[2] := '';
	END_IF
    
	//sValue3	
	IF fbMQTT_Values.axMatchFound[_Domoticz_eMQTT_PropertyNames.SValue3] THEN
		scMQTT_ObjectData_int.asValue[3] := fbMQTT_Values.asPropertyValue[_Domoticz_eMQTT_PropertyNames.SValue3];
	ELSE
		scMQTT_ObjectData_int.asValue[3] := '';
	END_IF
	
    //sValue4	
	IF fbMQTT_Values.axMatchFound[_Domoticz_eMQTT_PropertyNames.SValue4] THEN
		scMQTT_ObjectData_int.asValue[4] := fbMQTT_Values.asPropertyValue[_Domoticz_eMQTT_PropertyNames.SValue4];
	ELSE
		scMQTT_ObjectData_int.asValue[4] := '';
	END_IF
	
    //sValue5	
	IF fbMQTT_Values.axMatchFound[_Domoticz_eMQTT_PropertyNames.SValue5] THEN
		scMQTT_ObjectData_int.asValue[5] := fbMQTT_Values.asPropertyValue[_Domoticz_eMQTT_PropertyNames.SValue5];
	ELSE
		scMQTT_ObjectData_int.asValue[5] := '';
	END_IF
	
	//sValue6    
	IF fbMQTT_Values.axMatchFound[_Domoticz_eMQTT_PropertyNames.SValue6] THEN
		scMQTT_ObjectData_int.asValue[6] := fbMQTT_Values.asPropertyValue[_Domoticz_eMQTT_PropertyNames.SValue6];
	ELSE
		scMQTT_ObjectData_int.asValue[6] := '';
	END_IF
	
	//Color (R)    
	IF fbMQTT_Values.axMatchFound[_Domoticz_eMQTT_PropertyNames.ColorR] THEN
		scMQTT_ObjectData_int.asValue[Domoticz_eSValues_Colors.Red] := fbMQTT_Values.asPropertyValue[_Domoticz_eMQTT_PropertyNames.ColorR];
	END_IF
	//Color (G)    
	IF fbMQTT_Values.axMatchFound[_Domoticz_eMQTT_PropertyNames.ColorG] THEN
		scMQTT_ObjectData_int.asValue[Domoticz_eSValues_Colors.Green] := fbMQTT_Values.asPropertyValue[_Domoticz_eMQTT_PropertyNames.ColorG];
	END_IF
	//Color (B)    
	IF fbMQTT_Values.axMatchFound[_Domoticz_eMQTT_PropertyNames.ColorB] THEN
		scMQTT_ObjectData_int.asValue[Domoticz_eSValues_Colors.Blue] := fbMQTT_Values.asPropertyValue[_Domoticz_eMQTT_PropertyNames.ColorB];
	END_IF
	//Color (CW)    
	IF fbMQTT_Values.axMatchFound[_Domoticz_eMQTT_PropertyNames.ColorCW] THEN
		scMQTT_ObjectData_int.asValue[Domoticz_eSValues_Colors.ColdWhite] := fbMQTT_Values.asPropertyValue[_Domoticz_eMQTT_PropertyNames.ColorCW];
	END_IF
	//Color (WW)    
	IF fbMQTT_Values.axMatchFound[_Domoticz_eMQTT_PropertyNames.ColorWW] THEN
		scMQTT_ObjectData_int.asValue[Domoticz_eSValues_Colors.WarmWhite] := fbMQTT_Values.asPropertyValue[_Domoticz_eMQTT_PropertyNames.ColorWW];
	END_IF	
	//Brighness is a sValue1 > So automatically placed correctly
	
	//Adjust incoming values for P1 Smart meter (Energy)
	IF fbMQTT_Values.axMatchFound[_Domoticz_eMQTT_PropertyNames.SwitchType]
	AND fbMQTT_Values.asPropertyValue[_Domoticz_eMQTT_PropertyNames.SwitchType] = Domoticz_Constants.sType_Energy THEN
		scMQTT_ObjectData_int.asValue[Domoticz_eSValues_P1.Usage1Cumulative] := TO_STRING(TO_REAL(scMQTT_ObjectData_int.asValue[Domoticz_eSValues_P1.Usage1Cumulative])/1000.0);
		scMQTT_ObjectData_int.asValue[Domoticz_eSValues_P1.Usage2Cumulative] := TO_STRING(TO_REAL(scMQTT_ObjectData_int.asValue[Domoticz_eSValues_P1.Usage2Cumulative])/1000.0);
		scMQTT_ObjectData_int.asValue[Domoticz_eSValues_P1.Return1Cumulative] := TO_STRING(TO_REAL(scMQTT_ObjectData_int.asValue[Domoticz_eSValues_P1.Return1Cumulative])/1000.0);
		scMQTT_ObjectData_int.asValue[Domoticz_eSValues_P1.Return2Cumulative] := TO_STRING(TO_REAL(scMQTT_ObjectData_int.asValue[Domoticz_eSValues_P1.Return2Cumulative])/1000.0);
	//Adjust incoming values for Energy meter (kWh)
	ELSIF fbMQTT_Values.axMatchFound[_Domoticz_eMQTT_PropertyNames.SwitchType]
	AND fbMQTT_Values.asPropertyValue[_Domoticz_eMQTT_PropertyNames.SwitchType] = Domoticz_Constants.sType_kWh THEN
		scMQTT_ObjectData_int.asValue[Domoticz_eSValues_P1.Usage2Cumulative] := TO_STRING(TO_REAL(scMQTT_ObjectData_int.asValue[Domoticz_eSValues_P1.Usage2Cumulative])/1000.0);
	//Adjust incoming values for Gas meter (Gas)
	ELSIF fbMQTT_Values.axMatchFound[_Domoticz_eMQTT_PropertyNames.SwitchType]
	AND fbMQTT_Values.asPropertyValue[_Domoticz_eMQTT_PropertyNames.SwitchType] = Domoticz_Constants.sType_Gas THEN
		scMQTT_ObjectData_int.asValue[Domoticz_eSValues_P1.Usage1Cumulative] := TO_STRING(TO_REAL(scMQTT_ObjectData_int.asValue[Domoticz_eSValues_P1.Usage1Cumulative])/1000.0);
	END_IF
	
	//Adjust incoming values for Humidity
	//Round humidity
	IF fbMQTT_Values.asPropertyValue[_Domoticz_eMQTT_PropertyNames.ObjectType] = Domoticz_Constants.sType_TemperatureHumidity
	OR fbMQTT_Values.asPropertyValue[_Domoticz_eMQTT_PropertyNames.ObjectType] = Domoticz_Constants.sType_TemperatureHumidityBaro THEN
		IF (_Domoticz_StringToReal(scMQTT_ObjectData_int.asValue[Domoticz_eSValues_TempHumBaro.Humidity])
		- TO_REAL(TRUNC(_Domoticz_StringToReal(scMQTT_ObjectData_int.asValue[Domoticz_eSValues_TempHumBaro.Humidity])))) <= 0.5 THEN
			scMQTT_ObjectData_int.asValue[Domoticz_eSValues_TempHumBaro.Humidity] := TO_STRING(TRUNC(_Domoticz_StringToReal(scMQTT_ObjectData_int.asValue[Domoticz_eSValues_TempHumBaro.Humidity])));
		ELSIF (_Domoticz_StringToReal(scMQTT_ObjectData_int.asValue[Domoticz_eSValues_TempHumBaro.Humidity])
		- TO_REAL(TRUNC(_Domoticz_StringToReal(scMQTT_ObjectData_int.asValue[Domoticz_eSValues_TempHumBaro.Humidity])))) > 0.5 THEN
			scMQTT_ObjectData_int.asValue[Domoticz_eSValues_TempHumBaro.Humidity] := TO_STRING(TRUNC(_Domoticz_StringToReal(scMQTT_ObjectData_int.asValue[Domoticz_eSValues_TempHumBaro.Humidity]))+1);
		END_IF
	END_IF

	//Add info
	scMQTT_ObjectData_int.sDeviceType := fbMQTT_Values.asPropertyValue[_Domoticz_eMQTT_PropertyNames.ObjectType];	//Transfer type
	scMQTT_ObjectData_int.dtLastUpdate := scConnector.scTwilightData.dtSystem;		//Latest update is equal to timestamp (act time) in case of MQTT
	scMQTT_ObjectData_int.dtTimeStamp := scConnector.scTwilightData.dtSystem;
	scMQTT_ObjectData_int.eSource := _Domoticz_eDataSource.MQTT;
	
	//Round decimals
	FOR wX := 1 TO Domoticz_Constants.uiMaxSValues DO
		IF scMQTT_ObjectData_int.asValue[wX] <> '' THEN
			scMQTT_ObjectData_int.asValue[wX] := TO_STRING(_Domoticz_RoundDecimals(TO_REAL(scMQTT_ObjectData_int.asValue[wX]),2));
		END_IF
	END_FOR
	
	//Output data
	xMQTT_NewObject := TRUE;
	
	//Statistics
	udiUpdateRate_MQTT_int := udiUpdateRate_MQTT_int + 1;	//Update statistics
END_IF
END_ACTION

ACTION MQTT_DataObject_Out:
{attribute 'conditionalshow'}

//Get pointers
psMQTT_Concat := ADR(sMQTT_Concat);
psMQTT_ConcatHelper := ADR(sMQTT_ConcatHelper);


//Wait for new message
IF fbMQTT_Send.xConnected AND NOT fbMQTT_Send.xPublish //Connected and not busy yet
AND scConnector.xNewObject_Tx AND scConnector.scObjectData_Tx.uiIdentifier > 0 THEN	//New object placed and valid	
	sMQTT_Concat := '';//Reset message
	
	//Add start of JSON message
	sMQTT_ConcatHelper := '{';
	StrConcatA(psMQTT_ConcatHelper, psMQTT_Concat, TO_INT(SNDLTN_MQTT.MQTT_Properties.uiMQTTMaxMessageSize));
	
	//Add identifier start
	StrConcatA(ADR(Domoticz_Constants.sCommandMQTT_idx), psMQTT_Concat, TO_INT(SNDLTN_MQTT.MQTT_Properties.uiMQTTMaxMessageSize));
	
	//Add idx
	sMQTT_ConcatHelper := TO_STRING(scConnector.scObjectData_Tx.uiIdentifier);
	StrConcatA(psMQTT_ConcatHelper, psMQTT_Concat, TO_INT(SNDLTN_MQTT.MQTT_Properties.uiMQTTMaxMessageSize));
	
	//Close part
	sMQTT_ConcatHelper := ', ';
	StrConcatA(psMQTT_ConcatHelper, psMQTT_Concat, TO_INT(SNDLTN_MQTT.MQTT_Properties.uiMQTTMaxMessageSize));
	
	
	//Add command and values
	CASE scConnector.scObjectData_Tx.eCommand OF
		//All custom n-/s-value devices
		_Domoticz_eCommandType.Default:
		
			//Add command type
			StrConcatA(ADR(Domoticz_Constants.sCommandMQTT_uDevice), psMQTT_Concat, TO_INT(SNDLTN_MQTT.MQTT_Properties.uiMQTTMaxMessageSize));
			
			//Close part
			sMQTT_ConcatHelper := ', ';
			StrConcatA(psMQTT_ConcatHelper, psMQTT_Concat, TO_INT(SNDLTN_MQTT.MQTT_Properties.uiMQTTMaxMessageSize));
			
			//Add sValues if needed
			iCountMQTT_sValues := 0;
			FOR wX := 1 TO Domoticz_Constants.uiMaxSValues DO
				//Check object
				IF scConnector.scObjectData_Tx.asValue[wX] <> '' THEN
					//Add start / separator
					IF iCountMQTT_sValues = 0 THEN	//First element
						StrConcatA(ADR(Domoticz_Constants.sCommandMQTT_sValues), psMQTT_Concat, TO_INT(SNDLTN_MQTT.MQTT_Properties.uiMQTTMaxMessageSize));
					ELSE	//Already added svalue string, use separator
						sMQTT_ConcatHelper := ';';
						StrConcatA(psMQTT_ConcatHelper, psMQTT_Concat, TO_INT(SNDLTN_MQTT.MQTT_Properties.uiMQTTMaxMessageSize));
					END_IF
					//Add value
					sMQTT_ConcatHelper := scConnector.scObjectData_Tx.asValue[wX];
					StrConcatA(psMQTT_ConcatHelper, psMQTT_Concat, TO_INT(SNDLTN_MQTT.MQTT_Properties.uiMQTTMaxMessageSize));
					//Count object if used
					iCountMQTT_sValues := iCountMQTT_sValues + 1;
				END_IF
			END_FOR
			
			//Add closing marks if svalue has been used
			IF iCountMQTT_sValues > 0 THEN
				sMQTT_ConcatHelper := '", ';
				StrConcatA(psMQTT_ConcatHelper, psMQTT_Concat, TO_INT(SNDLTN_MQTT.MQTT_Properties.uiMQTTMaxMessageSize));
			END_IF
			
			//nValue
			//Add start
			StrConcatA(ADR(Domoticz_Constants.sCommandMQTT_nValue), psMQTT_Concat, TO_INT(SNDLTN_MQTT.MQTT_Properties.uiMQTTMaxMessageSize));
			
			sMQTT_ConcatHelper := TO_STRING(scConnector.scObjectData_Tx.iValue);
			StrConcatA(psMQTT_ConcatHelper, psMQTT_Concat, TO_INT(SNDLTN_MQTT.MQTT_Properties.uiMQTTMaxMessageSize));//Last element, no comma
		
		//Lights/switches
		_Domoticz_eCommandType.SwitchLight:
			//Add command type
			StrConcatA(ADR(Domoticz_Constants.sCommandMQTT_SwitchLight), psMQTT_Concat, TO_INT(SNDLTN_MQTT.MQTT_Properties.uiMQTTMaxMessageSize));
			
			//Close part
			sMQTT_ConcatHelper := ', ';
			StrConcatA(psMQTT_ConcatHelper, psMQTT_Concat, TO_INT(SNDLTN_MQTT.MQTT_Properties.uiMQTTMaxMessageSize));
			
			//Check value 
			CASE scConnector.scObjectData_Tx.iValue OF
				0:
				StrConcatA(ADR(Domoticz_Constants.sCommandMQTT_SwitchOff), psMQTT_Concat, TO_INT(SNDLTN_MQTT.MQTT_Properties.uiMQTTMaxMessageSize));
				
				1:
				StrConcatA(ADR(Domoticz_Constants.sCommandMQTT_SwitchOn), psMQTT_Concat, TO_INT(SNDLTN_MQTT.MQTT_Properties.uiMQTTMaxMessageSize));
				
				ELSE
				StrConcatA(ADR(Domoticz_Constants.sCommandMQTT_SwitchLevel), psMQTT_Concat, TO_INT(SNDLTN_MQTT.MQTT_Properties.uiMQTTMaxMessageSize));	
				
				//Close command
				sMQTT_ConcatHelper := ', ';
				StrConcatA(psMQTT_ConcatHelper, psMQTT_Concat, TO_INT(SNDLTN_MQTT.MQTT_Properties.uiMQTTMaxMessageSize));
				
				//Add level
				StrConcatA(ADR(Domoticz_Constants.sCommandMQTT_Level), psMQTT_Concat, TO_INT(SNDLTN_MQTT.MQTT_Properties.uiMQTTMaxMessageSize));	
				
				sMQTT_ConcatHelper := scConnector.scObjectData_Tx.asValue[1];
				StrConcatA(psMQTT_ConcatHelper, psMQTT_Concat, TO_INT(SNDLTN_MQTT.MQTT_Properties.uiMQTTMaxMessageSize));
				
			END_CASE
		
		//Scenes
		_Domoticz_eCommandType.SwitchScene:
			//Add command type
			StrConcatA(ADR(Domoticz_Constants.sCommandMQTT_SwitchScene), psMQTT_Concat, TO_INT(SNDLTN_MQTT.MQTT_Properties.uiMQTTMaxMessageSize));
			
			//Close part
			sMQTT_ConcatHelper := ', ';
			StrConcatA(psMQTT_ConcatHelper, psMQTT_Concat, TO_INT(SNDLTN_MQTT.MQTT_Properties.uiMQTTMaxMessageSize));
			//To be done
		
		//Color
		//{"command":"setcolbrightnessvalue", "idx":107, "color":{"m":3,"t":0,"r":255,"g":0,"b":0,"cw":0,"ww":0}}
		_Domoticz_eCommandType.SetColor:
			//Add command type
			StrConcatA(ADR(Domoticz_Constants.sCommandMQTT_Color), psMQTT_Concat, TO_INT(SNDLTN_MQTT.MQTT_Properties.uiMQTTMaxMessageSize));
			
			//Close part
			sMQTT_ConcatHelper := ', ';
			StrConcatA(psMQTT_ConcatHelper, psMQTT_Concat, TO_INT(SNDLTN_MQTT.MQTT_Properties.uiMQTTMaxMessageSize));
			
			//Add color values start
			StrConcatA(ADR(Domoticz_Constants.sCommandMQTT_Color_Value), psMQTT_Concat, TO_INT(SNDLTN_MQTT.MQTT_Properties.uiMQTTMaxMessageSize));
			
			//Add opening
			sMQTT_ConcatHelper := '{"';
			StrConcatA(psMQTT_ConcatHelper, psMQTT_Concat, TO_INT(SNDLTN_MQTT.MQTT_Properties.uiMQTTMaxMessageSize));
			
			
			//M (mode)
			StrConcatA(ADR(Domoticz_Constants.sCommandMQTT_Color_Mode), psMQTT_Concat, TO_INT(SNDLTN_MQTT.MQTT_Properties.uiMQTTMaxMessageSize));
			//Seperator
			sMQTT_ConcatHelper := '":';
			StrConcatA(psMQTT_ConcatHelper, psMQTT_Concat, TO_INT(SNDLTN_MQTT.MQTT_Properties.uiMQTTMaxMessageSize));
			
			
			//ColorModeWhite = 1,  // White. Valid fields:none
			//ColorModeTemp = 2,   // White with color temperature. Valid fields:t
			//ColorModeRGB = 3,    // Color. Valid fields:r, g, b.
			//ColorModeCustom = 4, // Custom (color + white). Valid fields:r, g, b, cw, ww, depending on device capabilities
			
			//White (cold/warm)
			IF TO_REAL(scConnector.scObjectData_Tx.asValue[Domoticz_eSValues_Colors.ColdWhite]) > 0
			OR TO_REAL(scConnector.scObjectData_Tx.asValue[Domoticz_eSValues_Colors.WarmWhite]) > 0 THEN
				sMQTT_ConcatHelper := '2';
				StrConcatA(psMQTT_ConcatHelper, psMQTT_Concat, TO_INT(SNDLTN_MQTT.MQTT_Properties.uiMQTTMaxMessageSize));
			
			//Color
			ELSE
				sMQTT_ConcatHelper := '3';
				StrConcatA(psMQTT_ConcatHelper, psMQTT_Concat, TO_INT(SNDLTN_MQTT.MQTT_Properties.uiMQTTMaxMessageSize));
			
			//Custom mode is not supported by HUE / Milight, so no need for it
			END_IF

			//R (red)
			//Close previous
			sMQTT_ConcatHelper := ',"';
			StrConcatA(psMQTT_ConcatHelper, psMQTT_Concat, TO_INT(SNDLTN_MQTT.MQTT_Properties.uiMQTTMaxMessageSize));
			//Add command
			StrConcatA(ADR(Domoticz_Constants.asProperty_Colors[Domoticz_eSValues_Colors.Red]), psMQTT_Concat, TO_INT(SNDLTN_MQTT.MQTT_Properties.uiMQTTMaxMessageSize));
			//Seperate
			sMQTT_ConcatHelper := '":';
			StrConcatA(psMQTT_ConcatHelper, psMQTT_Concat, TO_INT(SNDLTN_MQTT.MQTT_Properties.uiMQTTMaxMessageSize));
			//Add value
			sMQTT_ConcatHelper := TO_STRING(TO_INT(scConnector.scObjectData_Tx.asValue[Domoticz_eSValues_Colors.Red]));
			StrConcatA(psMQTT_ConcatHelper, psMQTT_Concat, TO_INT(SNDLTN_MQTT.MQTT_Properties.uiMQTTMaxMessageSize));
			
			//G (green)
			//Close previous
			sMQTT_ConcatHelper := ',"';
			StrConcatA(psMQTT_ConcatHelper, psMQTT_Concat, TO_INT(SNDLTN_MQTT.MQTT_Properties.uiMQTTMaxMessageSize));
			//Add command
			StrConcatA(ADR(Domoticz_Constants.asProperty_Colors[Domoticz_eSValues_Colors.Green]), psMQTT_Concat, TO_INT(SNDLTN_MQTT.MQTT_Properties.uiMQTTMaxMessageSize));
			//Seperate
			sMQTT_ConcatHelper := '":';
			StrConcatA(psMQTT_ConcatHelper, psMQTT_Concat, TO_INT(SNDLTN_MQTT.MQTT_Properties.uiMQTTMaxMessageSize));
			//Add value
			sMQTT_ConcatHelper := TO_STRING(TO_INT(scConnector.scObjectData_Tx.asValue[Domoticz_eSValues_Colors.Green]));
			StrConcatA(psMQTT_ConcatHelper, psMQTT_Concat, TO_INT(SNDLTN_MQTT.MQTT_Properties.uiMQTTMaxMessageSize));
			
			//B (blue)
			//Close previous
			sMQTT_ConcatHelper := ',"';
			StrConcatA(psMQTT_ConcatHelper, psMQTT_Concat, TO_INT(SNDLTN_MQTT.MQTT_Properties.uiMQTTMaxMessageSize));
			//Add command
			StrConcatA(ADR(Domoticz_Constants.asProperty_Colors[Domoticz_eSValues_Colors.Blue]), psMQTT_Concat, TO_INT(SNDLTN_MQTT.MQTT_Properties.uiMQTTMaxMessageSize));
			//Seperate
			sMQTT_ConcatHelper := '":';
			StrConcatA(psMQTT_ConcatHelper, psMQTT_Concat, TO_INT(SNDLTN_MQTT.MQTT_Properties.uiMQTTMaxMessageSize));
			//Add value
			sMQTT_ConcatHelper := TO_STRING(TO_INT(scConnector.scObjectData_Tx.asValue[Domoticz_eSValues_Colors.Blue]));
			StrConcatA(psMQTT_ConcatHelper, psMQTT_Concat, TO_INT(SNDLTN_MQTT.MQTT_Properties.uiMQTTMaxMessageSize));
			
			//CW (cold white)
			//Close previous
			sMQTT_ConcatHelper := ',"';
			StrConcatA(psMQTT_ConcatHelper, psMQTT_Concat, TO_INT(SNDLTN_MQTT.MQTT_Properties.uiMQTTMaxMessageSize));
			//Add command
			StrConcatA(ADR(Domoticz_Constants.asProperty_Colors[Domoticz_eSValues_Colors.ColdWhite]), psMQTT_Concat, TO_INT(SNDLTN_MQTT.MQTT_Properties.uiMQTTMaxMessageSize));
			//Seperate
			sMQTT_ConcatHelper := '":';
			StrConcatA(psMQTT_ConcatHelper, psMQTT_Concat, TO_INT(SNDLTN_MQTT.MQTT_Properties.uiMQTTMaxMessageSize));
			//Add value
			sMQTT_ConcatHelper := TO_STRING(TO_INT(scConnector.scObjectData_Tx.asValue[Domoticz_eSValues_Colors.ColdWhite]));
			StrConcatA(psMQTT_ConcatHelper, psMQTT_Concat, TO_INT(SNDLTN_MQTT.MQTT_Properties.uiMQTTMaxMessageSize));			//Custom mode (4) not supported, value added anyway
			
			//WW (warm white)
			//Close previous
			sMQTT_ConcatHelper := ',"';
			StrConcatA(psMQTT_ConcatHelper, psMQTT_Concat, TO_INT(SNDLTN_MQTT.MQTT_Properties.uiMQTTMaxMessageSize));
			//Add command
			StrConcatA(ADR(Domoticz_Constants.asProperty_Colors[Domoticz_eSValues_Colors.WarmWhite]), psMQTT_Concat, TO_INT(SNDLTN_MQTT.MQTT_Properties.uiMQTTMaxMessageSize));
			//Seperate
			sMQTT_ConcatHelper := '":';
			StrConcatA(psMQTT_ConcatHelper, psMQTT_Concat, TO_INT(SNDLTN_MQTT.MQTT_Properties.uiMQTTMaxMessageSize));
			//Add value
			sMQTT_ConcatHelper := TO_STRING(TO_INT(scConnector.scObjectData_Tx.asValue[Domoticz_eSValues_Colors.WarmWhite]));
			StrConcatA(psMQTT_ConcatHelper, psMQTT_Concat, TO_INT(SNDLTN_MQTT.MQTT_Properties.uiMQTTMaxMessageSize));		//Custom mode (4) not supported, value added anyway
			
			//T (temperature)
			//Close previous
			sMQTT_ConcatHelper := ',"';
			StrConcatA(psMQTT_ConcatHelper, psMQTT_Concat, TO_INT(SNDLTN_MQTT.MQTT_Properties.uiMQTTMaxMessageSize));
			//Add command
			StrConcatA(ADR(Domoticz_Constants.sCommandMQTT_Color_Temperature), psMQTT_Concat, TO_INT(SNDLTN_MQTT.MQTT_Properties.uiMQTTMaxMessageSize));
			//Seperate
			sMQTT_ConcatHelper := '":';
			StrConcatA(psMQTT_ConcatHelper, psMQTT_Concat, TO_INT(SNDLTN_MQTT.MQTT_Properties.uiMQTTMaxMessageSize));

			//Add calculated temperature value
			IF TO_BYTE(scConnector.scObjectData_Tx.asValue[Domoticz_eSValues_Colors.WarmWhite]) > 0
			OR TO_BYTE(scConnector.scObjectData_Tx.asValue[Domoticz_eSValues_Colors.ColdWhite]) > 0 THEN
				rMQTT_ColorTemperature := LIMIT(0,(128 + TO_REAL(scConnector.scObjectData_Tx.asValue[Domoticz_eSValues_Colors.WarmWhite]) - TO_REAL(scConnector.scObjectData_Tx.asValue[Domoticz_eSValues_Colors.ColdWhite])), 255);
			ELSE
				rMQTT_ColorTemperature := 0.0;
			END_IF
			sMQTT_ConcatHelper := TO_STRING(TO_INT(rMQTT_ColorTemperature));
			StrConcatA(psMQTT_ConcatHelper, psMQTT_Concat, TO_INT(SNDLTN_MQTT.MQTT_Properties.uiMQTTMaxMessageSize));
			
			//Close off
			sMQTT_ConcatHelper := '}';
			StrConcatA(psMQTT_ConcatHelper, psMQTT_Concat, TO_INT(SNDLTN_MQTT.MQTT_Properties.uiMQTTMaxMessageSize));
			
			//Close command
			sMQTT_ConcatHelper := ', ';
			StrConcatA(psMQTT_ConcatHelper, psMQTT_Concat, TO_INT(SNDLTN_MQTT.MQTT_Properties.uiMQTTMaxMessageSize));
			
			//Add brightness
			StrConcatA(ADR(Domoticz_Constants.sCommandMQTT_Brightness), psMQTT_Concat, TO_INT(SNDLTN_MQTT.MQTT_Properties.uiMQTTMaxMessageSize));	
			
			sMQTT_ConcatHelper := TO_STRING(TO_INT(scConnector.scObjectData_Tx.asValue[Domoticz_eSValues_Colors.Brightness]));
			StrConcatA(psMQTT_ConcatHelper, psMQTT_Concat, TO_INT(SNDLTN_MQTT.MQTT_Properties.uiMQTTMaxMessageSize));

			
		//Brightness
		//{"command":"switchlight", "idx":107, "switchcmd":"Set Level", "level":10}
		_Domoticz_eCommandType.SetBrightness:
			//Add command type
			StrConcatA(ADR(Domoticz_Constants.sCommandMQTT_SwitchLight), psMQTT_Concat, TO_INT(SNDLTN_MQTT.MQTT_Properties.uiMQTTMaxMessageSize));
			
			//Close part
			sMQTT_ConcatHelper := ', ';
			StrConcatA(psMQTT_ConcatHelper, psMQTT_Concat, TO_INT(SNDLTN_MQTT.MQTT_Properties.uiMQTTMaxMessageSize));
			
			//Add command
			StrConcatA(ADR(Domoticz_Constants.sCommandMQTT_SwitchLevel), psMQTT_Concat, TO_INT(SNDLTN_MQTT.MQTT_Properties.uiMQTTMaxMessageSize));	
			
			//Close command
			sMQTT_ConcatHelper := ', ';
			StrConcatA(psMQTT_ConcatHelper, psMQTT_Concat, TO_INT(SNDLTN_MQTT.MQTT_Properties.uiMQTTMaxMessageSize));
			
			//Add level
			StrConcatA(ADR(Domoticz_Constants.sCommandMQTT_Level), psMQTT_Concat, TO_INT(SNDLTN_MQTT.MQTT_Properties.uiMQTTMaxMessageSize));	
			
			sMQTT_ConcatHelper := TO_STRING(TO_INT(scConnector.scObjectData_Tx.asValue[Domoticz_eSValues_Colors.Brightness]));
			StrConcatA(psMQTT_ConcatHelper, psMQTT_Concat, TO_INT(SNDLTN_MQTT.MQTT_Properties.uiMQTTMaxMessageSize));
		
	END_CASE
	
	//Add end of message
	sMQTT_ConcatHelper := '}';
	StrConcatA(psMQTT_ConcatHelper, psMQTT_Concat, TO_INT(SNDLTN_MQTT.MQTT_Properties.uiMQTTMaxMessageSize));
		
	//Transfer
	fbMQTT_Send.sPublishMessage := sMQTT_Concat;
	
	//Send message
	fbMQTT_Send.xPublish := TRUE;

//Wait until done
ELSIF (scConnector.xNewObject_Tx AND fbMQTT_Send.xPublish AND fbMQTT_Send.xPublished ) //New object published
OR (scConnector.xNewObject_Tx AND scConnector.scObjectData_Tx.uiIdentifier = 0) //New object not valid
OR TON_MQTT_PublishTimeout.Q THEN //Timeout publishing
	scConnector.xNewObject_Tx := FALSE;	//Make room for new update
	scConnector.scObjectData_Tx := scObjectData_Empty; //Empty
	fbMQTT_Send.xPublish := FALSE;
END_IF

//Give data time to be processed
TON_MQTT_PublishTimeout(IN:=fbMQTT_Send.xPublish, PT:=T#100MS);
END_ACTION

ACTION SystemTime:
{attribute 'conditionalshow'}

//System time

//Get time
TP_SysTime(IN:= NOT FB_SysTime_Get.xExecute, PT:= T#500MS);
FB_SysTime_Get(xExecute:= TP_SysTime.Q);
//Transfer time
IF FB_SysTime_Get.xDone 
AND FB_SysTime_Get.dtDateAndTime <> DT#1970-1-1-0:0:0 THEN 
	scConnector.scTwilightData.dtSystem := FB_SysTime_Get.dtDateAndTime; 
END_IF
scConnector.scTwilightData.todSystem := DT_TO_TOD(scConnector.scTwilightData.dtSystem);

//Set time
udiSysTime_Set := TO_UDINT(scConnector.scTwilightData.dtServer) + TO_UDINT(TO_DT(todSystemTime_Offset_int));
FB_SysTime_Set(xExecute := xAutoSyncClocks_int 
						AND xSyncTime_int, 
				dtDateAndTime := TO_DT(udiSysTime_Set));
IF (FB_SysTime_Set.xDone AND xSyncTime_int) 
OR FB_SysTime_Set.xError THEN 
	xSyncTime_int := FALSE; 
END_IF	//Remove trigger when done or error

//Create pulses on specific times
//Other data is filled from HTTP_DataTwilight

//Astronomic
scConnector.scTwilightData.xAstronomicRise := scConnector.scTwilightData.todSystem = scConnector.scTwilightData.todAstronomicRise;
scConnector.scTwilightData.xAstronomicSet 	:= scConnector.scTwilightData.todSystem = scConnector.scTwilightData.todAstronomicSet;

//Nautic
scConnector.scTwilightData.xNauticRise 	:= scConnector.scTwilightData.todSystem = scConnector.scTwilightData.todNauticRise;
scConnector.scTwilightData.xNauticSet 		:= scConnector.scTwilightData.todSystem = scConnector.scTwilightData.todNauticSet;

//Civil
scConnector.scTwilightData.xCivilRise 		:= scConnector.scTwilightData.todSystem = scConnector.scTwilightData.todCivilRise;
scConnector.scTwilightData.xCivilSet 		:= scConnector.scTwilightData.todSystem = scConnector.scTwilightData.todCivilSet;

//Sun
scConnector.scTwilightData.xPreSunRise 	:= scConnector.scTwilightData.todSystem = scConnector.scTwilightData.todPreSunRise;
scConnector.scTwilightData.xSunRise 		:= scConnector.scTwilightData.todSystem = scConnector.scTwilightData.todSunRise;
scConnector.scTwilightData.xPostSunRise 	:= scConnector.scTwilightData.todSystem = scConnector.scTwilightData.todPostSunRise;
scConnector.scTwilightData.xPreSunSet 		:= scConnector.scTwilightData.todSystem = scConnector.scTwilightData.todPreSunSet;
scConnector.scTwilightData.xSunSet 		:= scConnector.scTwilightData.todSystem = scConnector.scTwilightData.todSunSet;
scConnector.scTwilightData.xPostSunSet 	:= scConnector.scTwilightData.todSystem = scConnector.scTwilightData.todPostSunSet;
scConnector.scTwilightData.xSunAtSouth 	:= scConnector.scTwilightData.todSystem = scConnector.scTwilightData.todSunAtSouth;

